// TwinCAT 3 PLC project PDxxPLC
// Title: PDxx
// Company: iMusic AS
// Author: Jakob Bak
// ProjectVersion: 0.4.0.3
// Description: Library for using the Nanotec PDxx series Stepper Motor with Controller
// ProgramVersion: 3.1.4024.0
// libraries:
//   Tc2_Standard, * (Beckhoff Automation GmbH)
//   Tc2_System, * (Beckhoff Automation GmbH)
//   Tc3_Module, * (Beckhoff Automation GmbH)
// project tree:
//   DUTs/ E_PDxx_ErrorNumber.TcDUT, E_PDxx_ModesOfOperation.TcDUT, E_PDxx_State.TcDUT, E_PDxx_TransitionCommand.TcDUT, ST_CANopenDevice.TcDUT, ST_PDxx_ControlWord.TcDUT, ST_PDxx_ErrorRegister.TcDUT, ST_PDxx_IO.TcDUT, ST_PDxx_PredefinedErrorField.TcDUT, ST_PDxx_RxTxPDOs.TcDUT, ST_PDxx_SimulationParameters.TcDUT, ST_PDxx_Status.TcDUT, ST_PDxx_StatusWord.TcDUT
//   / PlcTask.TcTTO
//   POUs/ FB_PDxxSimulation.TcPOU, FB_PDxx.TcPOU, FB_SDO.TcPOU, MAIN.TcPOU, FB_PDxxTester.TcPOU
//   Version/ Global_Version.TcGVL
// real-time tasks:
//   TASK PlcTask: cycle T#10ms, priority 20, ADS port 350
// I/O:
//   DEVICE Device 2 (EtherCAT), AmsNetId 10.3.0.21.3.1
//     Term 1 (EK1100) [EK1100 EtherCAT Coupler (2A E-Bus)]
//       Term 2 (EL6751) [EL6751 CANopen Master]
//       Term 3 (EL9011) [EL9011 End Terminal]
//   DEVICE Device 1 (EL6751), AmsNetId 10.3.0.21.2.1
//     Box 1 (PD2-C411L18-E-65-08)
//     Box 2 (PD4-E601L42-E-65-2)
// variable links:
//   PDxxPLC Instance <-> Device 1 (EL6751)/Box 1 (PD2-C411L18-E-65-08)
//     PlcTask Inputs/MAIN.fbPDxxTester.PDxx.stPDOs.TxPDO_1_6041h_StatusWord <-> TxPDO 1/Inputs/Statusword
//     PlcTask Inputs/MAIN.fbPDxxTester.PDxx.stPDOs.TxPDO_1_6061h_ModesOfOperationDisplay <-> TxPDO 1/Inputs/Modes of operation display
//     PlcTask Inputs/MAIN.fbPDxxTester.PDxx.stPDOs.TxPDO_2_6064h_PositionActualValue <-> TxPDO 2/Inputs/Position actual value
//     PlcTask Inputs/MAIN.fbPDxxTester.PDxx.stPDOs.TxPDO_3_6044h_VelocityActualValue <-> TxPDO 3/Inputs/vl velocity actual value
//     PlcTask Inputs/MAIN.fbPDxxTester.PDxx.stPDOs.TxPDO_4_60FDh_DigitalInputs <-> TxPDO 4/Inputs/Digital Inputs
//     PlcTask Outputs/MAIN.fbPDxxTester.PDxx.stPDOs.RxPDO_1_3202h_MotorDriveSubmodeSelect <-> RxPDO 1/Outputs/Motor drive submode select
//     PlcTask Outputs/MAIN.fbPDxxTester.PDxx.stPDOs.RxPDO_1_6040h_ControlWord <-> RxPDO 1/Outputs/Controlword
//     PlcTask Outputs/MAIN.fbPDxxTester.PDxx.stPDOs.RxPDO_1_6060h_ModesOfOperation <-> RxPDO 1/Outputs/Modes of operation
//     PlcTask Outputs/MAIN.fbPDxxTester.PDxx.stPDOs.RxPDO_2_607Ah_TargetPosition <-> RxPDO 2/Outputs/Target Position
//     PlcTask Outputs/MAIN.fbPDxxTester.PDxx.stPDOs.RxPDO_2_6081h_ProfileVelocity <-> RxPDO 2/Outputs/Profile velocity
//     PlcTask Outputs/MAIN.fbPDxxTester.PDxx.stPDOs.RxPDO_3_6042h_TargetVelocity <-> RxPDO 3/Outputs/vl target velocity
//     PlcTask Outputs/MAIN.fbPDxxTester.PDxx.stPDOs.RxPDO_4_60FEh_DigitalOutputs <-> RxPDO 4/Outputs/Digital Outputs #1

CONFIGURATION PDxxPLC
    RESOURCE PLC ON TwinCAT3
        TASK PlcTask(INTERVAL := T#10ms, PRIORITY := 20);
        PROGRAM MAIN WITH PlcTask : MAIN;
    END_RESOURCE
END_CONFIGURATION

// ---- DUTs/E_PDxx_ErrorNumber.TcDUT
{attribute 'qualified_only'}
{attribute 'strict'}
TYPE E_PDxx_ErrorNumber :
(
	// The following is taken from the manual for the PD4-E(CANopen) section 1003h.
	// It pertains to the firmware version v1748, so other firmware versions and other types of motors may have different error number 
	WATCHDOG_RESET 						:= 0, // Watchdog-Reset
	INPUT_VOLTAGE_TOO_HIGH				:= 1, // Input voltage too high
	OUTPUT_CURRENT_TOO_HIGH 			:= 2, // Output current too high
	INPUT_VOLTAGE_TOO_LOW 				:= 3, // Input voltage too low
	ERROR_AT_FIELDBUS 					:= 4, // Error at fieldbus
	MOTOR_TURNS_WRONG_DIRECTION			:= 5, // Motor turns – in spite of active block – in the wrong direction
	NMT_MASTER_TAKES_TOO_LONG_TO_SEND	:= 6, // CANopen only: NMT master takes too long to send nodeguarding request
	ENCODER_ERROR_ELECTRICAL_FAULT		:= 7, // Encoder error due to electrical fault or defective hardware
	ENCODER_ERROR_INDEX_NOT_FOUND		:= 8, // Encoder error; index not found during the auto setup
	ERROR_IN_AB_TRACK					:= 9, // Error in the AB track
	POSITIVE_LIMIT_SWITCH_ZONE_EXCEEDED := 10, //  Positive limit switch and tolerance zone exceeded
	NEGATIVE_LIMIT_SWITCH_ZONE_EXCEEDED := 11, // Negative limit switch and tolerance zone exceeded
	DEVICE_TEMPERATURE_ERROR			:= 12, // Device temperature above 80°C
	FOLLOWING_ERROR_WINDOW_AND_TIMEOUT	:= 13, // The values of object 6065h (Following Error Window) and object 6066h (Following Error Time Out) were exceeded; a fault was triggered.
	NONVOLATIVE_MEMORY_FULL_FOURTEEN	:= 14, // Warning: Nonvolatile memory full; controller must be restarted for cleanup work.
	MOTOR_BLOCKED						:= 15, // Motor blocked
	NONVOLATIVE_MEMORY_DAMAGED			:= 16, // Warning: Nonvolatile memory damaged; controller must be restarted for cleanup work.
	SLAVE_TOOK_TOO_LONG_TO_SEND_PDO		:= 17, // CANopen only: Slave took too long TO send PDO messages.
	HALL_SENSOR_FAULTY					:= 18, // Hall sensor faulty
	PDO_NOT_PROCESSED_DUE_LENGTH_ERROR	:= 19, // CANopen only: PDO not processed due to a length error
	PDO_LENGTH_EXCEEDED					:= 20, // CANopen only: PDO length exceeded
	NONVOLATIVE_MEMORY_FULL_TWENTY_ONE	:= 21, // Warning: Nonvolatile memory full; controller must be restarted for cleanup work.
	RATED_CURRENT_MUST_BE_SET			:= 22, // Rated current must be set (203Bh:01h)
	ENCODER_RESOLUTION_SET_INCORRECTLY	:= 23, // Encoder resolution, number of pole pairs and some other values are incorrect.
	MOTOR_CURRENT_TOO_HIGH_ADJUST_PI	:= 24, // Motor current is too high, adjust the PI parameters.
	INTERNAL_SOFTWARE_ERROR				:= 25, // Internal software error, generic
	CURRENT_TOO_HIGH_AT_DIGITAL_OUTPUT	:= 26, // Current too high at digital output
	UNEXPECTED_SYNC_LENGTH				:= 27, // CANopen only: Unexpected sync length
	OP_SWITCH_WITHOUT_STOPPING_MOTOR	:= 28, // EtherCAT only: The motor was stopped because EtherCAT switched state from OP to either SafeOP or PreOP without first stopping the motor.
	SLIPPAGE_ERROR_TOO_LARGE			:= 30 // Error in speed monitoring: slippage error too large
);
END_TYPE

// ---- DUTs/E_PDxx_ModesOfOperation.TcDUT
{attribute 'qualified_only'}
{attribute 'strict'}
TYPE E_PDxx_ModesOfOperation :
(
	AUTO_SETUP := -2,
	CLOCK_DIRECTION_MODE,
	NO_MODE_CHANGE_OR_NO_MODE_ASSIGNED,
	PROFILE_POSITION_MODE,
	VELOCITY_MODE,
	PROFILE_VELOCITY_MODE,
	PROFILE_TORQUE_MODE,
	RESERVED,
	HOMING_MODE,
	INTERPOLATED_POSITION_MODE,
	CYCLIC_SYNCHRONOUS_POSITION_MODE,
	CYCLIC_SYNCHRONOUS_VELOCITY_MODE,
	CYCLIC_SYNCHRONOUS_TORQUE_MODE
);
END_TYPE

// ---- DUTs/E_PDxx_State.TcDUT
{attribute 'qualified_only'}
{attribute 'strict'}
TYPE E_PDxx_State :
(
	UNKNOWN_STATE, 
	NOT_READY_TO_SWITCH_ON, 
	SWITCH_ON_DISABLED, 
	READY_TO_SWITCH_ON, 
	SWITCHED_ON, 
	OPERATION_ENABLED, 
	QUICK_STOP_ACTIVE, 
	FAULT_REACTION_ACTIVE, 
	FAULT
);
END_TYPE

// ---- DUTs/E_PDxx_TransitionCommand.TcDUT
{attribute 'qualified_only'}
{attribute 'strict'}
TYPE E_PDxx_TransitionCommand :
(
	SHUTDOWN := 0,
	SWITCH_ON,
	DISABLE_VOLTAGE,
	QUICK_STOP,
	ENABLE_OPERATION,
	FAULT_RESET
);
END_TYPE

// ---- DUTs/ST_CANopenDevice.TcDUT
TYPE ST_CANopenDevice :
STRUCT
    AmsNetId	: STRING(23); (* The AMSNetID addresses the EL6751. Can be empty if only one local single channel card is present*)
    PortNr		: WORD;       (* This Port No. addresses the CANopen Node (see System Manager) *)
END_STRUCT
END_TYPE

// ---- DUTs/ST_PDxx_ControlWord.TcDUT
TYPE ST_PDxx_ControlWord :
STRUCT
	SwitchedOn_bit_0			: BOOL; // Value = "1": Switches to the "Switched on" state
	EnableVoltage_bit_1			: BOOL; // Value = "1": Switches to the "Enable voltage" state
	QuickStop_bit_2				: BOOL; // Value = "0": Switches to the "Quick stop" state
	EnableOperation_bit_3		: BOOL; // Value = "1": Switches to the "Enable operation" state
	OperationModeSpecific_bit_4	: BOOL; // Meaning is dependent on the selected operating mode
	OperationModeSpecific_bit_5	: BOOL; // Meaning is dependent on the selected operating mode
	OperationModeSpecific_bit_6	: BOOL; // Meaning is dependent on the selected operating mode
	FaultReset_bit_7			: BOOL; // Resets an error (if possible)
	Halt_bit_8					: BOOL; // Value = "1": Triggers a halt; valid in the following modes: Profile Position, Velocity, Profile Velocity, Profile Torque, Interpolated Position Mode
	OperationModeSpecific_bit_9	: BOOL; // not described in the manual...
	
	eState : E_PDxx_State;
END_STRUCT
END_TYPE

// ---- DUTs/ST_PDxx_ErrorRegister.TcDUT

TYPE ST_PDxx_ErrorRegister :
STRUCT
	// Taken from manual section "1001h Error Register"
	GEN : BIT; // bit 0 - General error
	CUR : BIT; // bit 1 - Current
	VOL : BIT; // bit 2 - Voltage
	TEMP: BIT; // bit 3 - Temperature
	COM : BIT; // bit 4 - Communication
	PROF: BIT; // bit 5 - Relates TO the device profile
	RES : BIT; // bit 6 - Reserved, always "0"
	MAN : BIT; // bit 7 - Manufacturer-specific: The motor turns in the wrong direction.
END_STRUCT
END_TYPE

// ---- DUTs/ST_PDxx_IO.TcDUT
TYPE ST_PDxx_IO :
STRUCT
(* These values can be read with PDO on 60FDh *)
	InputNegativeLimitSwitch		: BOOL;
	InputPositiveLimitSwitch		: BOOL;
	InputHomeSwitch					: BOOL;
	Input1		: BOOL;
	Input2		: BOOL;
	Input3		: BOOL;
	Input4		: BOOL;
	Input5		: BOOL;
	Input6		: BOOL;
	Input7		: BOOL;
	Input8		: BOOL;

(* The below values has to be read/set with SDO 3240h *)	
	InputNegativeLimitSwitchEnabled	: BOOL;
	InputPositiveLimitSwitchEnabled	: BOOL;
	InputHomeSwitchEnabled			: BOOL;
	Input1_Inverted	: BOOL;
	Input2_Inverted	: BOOL;
	Input3_Inverted	: BOOL;
	Input4_Inverted	: BOOL;
	Input5_Inverted	: BOOL;
	Input6_Inverted	: BOOL;
	Input7_Inverted	: BOOL;
	Input8_Inverted	: BOOL;
	Input1_24V		: BOOL;
	Input2_24V		: BOOL;
	Input3_24V		: BOOL;
	Input4_24V		: BOOL;
	Input5_24V		: BOOL;
	Input6_24V		: BOOL;
	Input7_24V		: BOOL;
	Input8_24V		: BOOL;

//	OutputBrake	: BOOL;
//	Output1		: BOOL;
//	Output2		: BOOL;
//	Output3		: BOOL;
//	Output4		: BOOL;
END_STRUCT
END_TYPE

// ---- DUTs/ST_PDxx_PredefinedErrorField.TcDUT

TYPE ST_PDxx_PredefinedErrorField :
STRUCT
	nErrorNumber	: USINT;
	stErrorClass	: ST_PDxx_ErrorRegister;
	nErrorCode		: UINT;
END_STRUCT
END_TYPE

// ---- DUTs/ST_PDxx_RxTxPDOs.TcDUT
TYPE ST_PDxx_RxTxPDOs :
STRUCT
	TxPDO_1_6041h_StatusWord					: UINT;
	TxPDO_1_6061h_ModesOfOperationDisplay		: SINT;
	TxPDO_2_6064h_PositionActualValue			: DINT;
	TxPDO_3_6044h_VelocityActualValue			: INT;
	TxPDO_4_60FDh_DigitalInputs					: UDINT;
	
	RxPDO_1_6040h_ControlWord					: UINT;
	RxPDO_1_6060h_ModesOfOperation				: SINT;
	RxPDO_1_3202h_MotorDriveSubmodeSelect		: UDINT;
	RxPDO_2_607Ah_TargetPosition				: DINT;
	RxPDO_2_6081h_ProfileVelocity				: UDINT;
	RxPDO_3_6042h_TargetVelocity				: INT;
	RxPDO_4_60FEh_DigitalOutputs				: UDINT;
END_STRUCT
END_TYPE

// ---- DUTs/ST_PDxx_SimulationParameters.TcDUT
TYPE ST_PDxx_SimulationParameters :
STRUCT
	bActivateSimulation		: BOOL := FALSE;
	nPositionMin			: LREAL := 0; // mm
	nPositionMax			: LREAL := 1000; // mm
	nSecondsPerSimStep 		: LREAL := 0.010; // seconds
	nMMPerSecondPerVelUnit	: LREAL := 0.1667; // mm/s, for example rpm at 10mm per revolution, is 10 mm per minute, and hence this value 10 / 60 = 0.16667.
	
	bObjectInserted			: BOOL;
	nObjectThickness		: LREAL := 0.0; // mm
END_STRUCT
END_TYPE

// ---- DUTs/ST_PDxx_Status.TcDUT
TYPE ST_PDxx_Status :
STRUCT
	bZeroInitialised 			: BOOL := FALSE;
	bReversePolarity			: BOOL;
	nHomePosition				: DINT;
	nCurrentPosition			: DINT;
	nCurrentVelocity			: INT;
	nTargetPosition				: DINT;
	nMinActualPosition			: DINT;
	nMaxActualPosition			: DINT;
	bHasError					: BOOL;
	stErrorRegister				: ST_PDxx_ErrorRegister;
	nNumErrors					: USINT;
	ErrorField					: ARRAY [1..8] OF ST_PDxx_PredefinedErrorField;
END_STRUCT
END_TYPE

// ---- DUTs/ST_PDxx_StatusWord.TcDUT
TYPE ST_PDxx_StatusWord :
STRUCT
	ReadyToSwitchOn		: BOOL; // Value = "1": Controller is in the "Ready to Switch On" state (dependent on other bits, see following bit mask)
	SwitchedOn 			: BOOL; // Value = "1": Controller is in the "Switched On" state (dependent on other bits, see following bit mask)
	OperationEnabled	: BOOL; // Value = "1": Controller is in the "Operation Enabled" state (dependent on other bits, see following bit mask)
	Fault				: BOOL; // Error occurred
	VoltageEnabled		: BOOL; // Voltage applied
	QuickStop			: BOOL; // Value = "0": Controller is in the "Quick Stop" state (dependent on other bits, see following bit mask)
	SwitchOnDisabled	: BOOL;	// Value = "1": Controller is in the "Switched On Disabled" state (dependent on other bits, see following bit mask)
	Warning				: BOOL;	// Value = "1": Warning
	Synchronization		: BOOL;	// Value = "1": Controller is in sync with the fieldbus; value = "0": Controller is not in sync with the fieldbus
	Remote				: BOOL;	// Remote (value of the bit is always "1")
	TargetReached		: BOOL; // Target reached
	InternalLimitReached: BOOL;	// Limit exceeded
	OperationModeSpecific_bit12: BOOL; // Meaning is dependent on the selected operating mode
	OperationModeSpecific_bit13: BOOL; // Meaning is dependent on the selected operating mode
	ClosedLoopAvailable	: BOOL; // Value = "1": Auto setup was successful and encoder index seen: closed loop mode possible
END_STRUCT
END_TYPE

// ---- Version/Global_Version.TcGVL
{attribute 'TcGenerated'}
{attribute 'no-analysis'}
{attribute 'linkalways'}
// This function has been automatically generated from the project information.
VAR_GLOBAL CONSTANT
	{attribute 'const_non_replaced'}
	stLibVersion_PDxx : ST_LibVersion := (iMajor := 0, iMinor := 4, iBuild := 0, iRevision := 3, nFlags := 1, sVersion := '0.4.0.3');
END_VAR

// ---- POUs/MAIN.TcPOU

PROGRAM MAIN
VAR
	fbPDxxTester : FB_PDxxTester;
	stCANopenDevice : ST_CANopenDevice := (AmsNetId:='10.3.0.21.2.1', PortNr := 16#1001);
END_VAR


fbPDxxTester(stCANopenDevice := stCANopenDevice);

END_PROGRAM

// ---- POUs/FB_PDxxTester.TcPOU

FUNCTION_BLOCK FB_PDxxTester
VAR_INPUT

	stCANopenDevice 	: ST_CANopenDevice;
//	SimParameters		: ST_PDxx_SimulationParameters;
//	bStandAloneTesting 	: BOOL 		:= FALSE;

	nTargetVelocity		: INT := 100;			// what unit ?
	nTargetPosition		: DINT := 0;		// what unit ?
	nTargetCurrent		: UDINT := 1000;	// mA ?
//	bExecuteMove		: BOOL  := FALSE;
	
	nFeedRate			: UDINT := 44533;
	nFeedRateDivisor	: UDINT	:= 2000;
	nZeroingMaxCurrent	: UDINT := 1000;
	bReversePolarity	: BOOL := FALSE;
	
	eMode : (NO_CHANGE := 0, RESET, HOME, POSITION, VELOCITY);
END_VAR

VAR_OUTPUT
//	bTargetPositionReceived: BOOL;
	eState				: E_PDxx_State;
	eModesOfOperation	: E_PDxx_ModesOfOperation;
	
	Status 				: ST_PDxx_Status;
	StateEntryTime		: TIME;
	bStateComplete		: BOOL;
END_VAR

VAR
	PDxx : FB_PDxx;
//	trExecute : R_TRIG;
	eLastMode 			: INT;
END_VAR


ExecuteState();

PDxx(
	stCANopenDevice := stCANopenDevice,
//	SimParameters := SimParameters,
//	bStandAloneTesting := bStandAloneTesting,
//	bStandAloneTestSendTarget := bExecuteMove,
//	bStandAloneTestSendTargetSuccess => bTargetPositionReceived,
	Status => Status
);

eState := PDxx.eState;
eModesOfOperation := PDxx.eModesOfOperation;


METHOD PRIVATE ExecuteState

IF eMode <> NO_CHANGE THEN
	IF eMode <> eLastMode THEN
		eLastMode := eMode;
		StateEntryTime := TIME();
		bStateComplete := FALSE;
	END_IF
	
//	trExecute(CLK := bExecuteMove);	
	
	CASE eMode OF

		RESET:
			M_Resetting();

		HOME:
			PDxx.ProbeActualPositionLimits(nTargetVelocity);

		POSITION:
//			IF trExecute.Q = TRUE THEN
				PDxx.GoToTargetPosition(nPosition := nTargetPosition, nVelocity := nTargetVelocity, nMaxCurrent := nTargetCurrent);		
//			END_IF

		VELOCITY:
//			IF trExecute.Q = TRUE THEN
				PDxx.GoToTargetVelocity(nVelocity := nTargetVelocity, nMaxCurrent := nTargetCurrent);		
//			END_IF		

	END_CASE
	
	IF bStateComplete THEN
		eMode := NO_CHANGE;
	END_IF

END_IF
END_METHOD


METHOD PRIVATE M_Resetting : BOOL
VAR
	bFeedRateSetpointReached 	: BOOL := FALSE;
	bMaxCurrentSetpointReached 	: BOOL := FALSE;
	bPolaritySetpointReached	: BOOL := FALSE;
END_VAR

IF PDxx.SetFeedRate(nFeedRate := nFeedRate, nDivisor := nFeedRateDivisor) THEN
	bFeedRateSetpointReached := TRUE;
END_IF

IF PDxx.fbSdoMaxCurrentValue = nZeroingMaxCurrent THEN
	bMaxCurrentSetpointReached := TRUE;
ELSE
	PDxx.SetMaxCurrent(nZeroingMaxCurrent);
END_IF

IF 	PDxx.IsPolarityReversed() = bReversePolarity THEN
	bPolaritySetpointReached := TRUE;
ELSE
	bPolaritySetpointReached := PDxx.SetReversePolarity(bReversePolarity);
END_IF

(* COMPLETE STATE *)
IF 	bFeedRateSetpointReached AND
	bMaxCurrentSetpointReached AND
	bPolaritySetpointReached THEN 
	IF PDxx.SwitchOnPowerToMotor() THEN
		bStateComplete := TRUE;
	END_IF
ELSE
	PDxx.SwitchOffPowerToMotor();
END_IF
END_METHOD

END_FUNCTION_BLOCK

// ---- POUs/FB_PDxx.TcPOU
FUNCTION_BLOCK FB_PDxx

VAR_INPUT
	SimParameters		: ST_PDxx_SimulationParameters;

	eState				: E_PDxx_State;
	eModesOfOperation	: E_PDxx_ModesOfOperation;

	bStandAloneTesting 				: BOOL 		:= FALSE;
	eStandAloneTestState			: E_PDxx_State;
	eStandAloneTestModesOfOperation	: E_PDxx_ModesOfOperation;
	bStandAloneTestSendTarget		: BOOL 		:= 0;
	
	stCANopenDevice : ST_CANopenDevice;

	fbSdoErrorRegister				: FB_SDO	:= (CO_Index:=16#1001, CO_SubIndex:=16#0, DataLength:=1, 	CO_Name:='Error Register', 			stCANopenDevice:=stCANopenDevice);
	fbSdoErrorRegisterValue 		: USINT;

	fbSdoNumberOfErrors				: FB_SDO	:= (CO_Index:=16#1003, CO_SubIndex:=16#0, DataLength:=1, 	CO_Name:='Number Of Errors', 		stCANopenDevice:=stCANopenDevice);
	fbSdoNumberOfErrorsValue 		: USINT;

	fbSdoErrorField_1				: FB_SDO	:= (CO_Index:=16#1003, CO_SubIndex:=16#1, DataLength:=4, 	CO_Name:='Standard Error Field 1', 	stCANopenDevice:=stCANopenDevice);
	fbSdoErrorField_2				: FB_SDO	:= (CO_Index:=16#1003, CO_SubIndex:=16#2, DataLength:=4, 	CO_Name:='Standard Error Field 2', 	stCANopenDevice:=stCANopenDevice);
	fbSdoErrorField_3				: FB_SDO	:= (CO_Index:=16#1003, CO_SubIndex:=16#3, DataLength:=4, 	CO_Name:='Standard Error Field 3', 	stCANopenDevice:=stCANopenDevice);
	fbSdoErrorField_4				: FB_SDO	:= (CO_Index:=16#1003, CO_SubIndex:=16#4, DataLength:=4, 	CO_Name:='Standard Error Field 4', 	stCANopenDevice:=stCANopenDevice);
	fbSdoErrorField_5				: FB_SDO	:= (CO_Index:=16#1003, CO_SubIndex:=16#5, DataLength:=4, 	CO_Name:='Standard Error Field 5', 	stCANopenDevice:=stCANopenDevice);
	fbSdoErrorField_6				: FB_SDO	:= (CO_Index:=16#1003, CO_SubIndex:=16#6, DataLength:=4, 	CO_Name:='Standard Error Field 6', 	stCANopenDevice:=stCANopenDevice);
	fbSdoErrorField_7				: FB_SDO	:= (CO_Index:=16#1003, CO_SubIndex:=16#7, DataLength:=4, 	CO_Name:='Standard Error Field 7', 	stCANopenDevice:=stCANopenDevice);
	fbSdoErrorField_8				: FB_SDO	:= (CO_Index:=16#1003, CO_SubIndex:=16#8, DataLength:=4, 	CO_Name:='Standard Error Field 8', 	stCANopenDevice:=stCANopenDevice);
	fbSdoErrorFieldValue			: ARRAY [1..8] OF UDINT;

	fbSdoMaxCurrent					: FB_SDO	:= (CO_Index:=16#2031, CO_SubIndex:=16#0, DataLength:=4, 	CO_Name:='Maximum Current', 		stCANopenDevice:=stCANopenDevice);
	fbSdoMaxCurrentValue 			: UDINT;

//	fbSdoPolarity					: FB_SDO	:= (CO_Index:=16#607E, CO_SubIndex:=16#0, DataLength:=1, 	CO_Name:='Polarity', 				stCANopenDevice:=fbEL6751);
//	fbSdoPolarityValue				: USINT;

	fbSdoSpecialFunctionEnable		: FB_SDO	:= (CO_Index:=16#3040, CO_SubIndex:=16#1, DataLength:=4, 	CO_Name:='Special Function Enable',	stCANopenDevice:=stCANopenDevice);
	fbSdoSpecialFunctionEnableValue	: UDINT;

	fbSdoFunctionInverted			: FB_SDO	:= (CO_Index:=16#3040, CO_SubIndex:=16#2, DataLength:=4, 	CO_Name:='Function Inverted',		stCANopenDevice:=stCANopenDevice);
	fbSdoFunctionInvertedValue		: UDINT;
	
	fbSdoInputRangeSelect			: FB_SDO	:= (CO_Index:=16#3040, CO_SubIndex:=16#6, DataLength:=4, 	CO_Name:='Input Range Select',		stCANopenDevice:=stCANopenDevice);
	fbSdoInputRangeSelectValue		: UDINT;
	
	fbSdoFeed						: FB_SDO	:= (CO_Index:=16#6092, CO_SubIndex:=16#1, DataLength:=4, 	CO_Name:='Feed', 					stCANopenDevice:=stCANopenDevice);
	fbSdoFeedValue					: UDINT;

	fbSdoShaftRevolutions			: FB_SDO	:= (CO_Index:=16#6092, CO_SubIndex:=16#2, DataLength:=4, 	CO_Name:='Shaft Revolutions', 		stCANopenDevice:=stCANopenDevice);
	fbSdoShaftRevolutionsValue		: UDINT;
	
	fbSdoEncoderIncrements			: FB_SDO	:= (CO_Index:=16#608F, CO_SubIndex:=16#1, DataLength:=4, 	CO_Name:='Encoder Increments', 		stCANopenDevice:=stCANopenDevice);
	fbSdoEncoderIncrementsValue		: UDINT;

	fbSdoMotorRevolutions			: FB_SDO	:= (CO_Index:=16#608F, CO_SubIndex:=16#2, DataLength:=4, 	CO_Name:='Motor Revolutions', 		stCANopenDevice:=stCANopenDevice);
	fbSdoMotorRevolutionsValue		: UDINT;
	
	fbSdoSIUnitPosition				: FB_SDO	:= (CO_Index:=16#60A8, CO_SubIndex:=16#0, DataLength:=4, 	CO_Name:='SI Unit Position', 		stCANopenDevice:=stCANopenDevice);
	fbSdoSIUnitPositionValue		: UDINT;
	
	fbSdoProfileAcceleration		: FB_SDO	:= (CO_Index:=16#6083, CO_SubIndex:=16#0, DataLength:=4, 	CO_Name:='Profile Acceleration', 	stCANopenDevice:=stCANopenDevice);
	fbSdoProfileAccelerationValue	: UDINT;

	fbSdoProfileDeceleration		: FB_SDO	:= (CO_Index:=16#6084, CO_SubIndex:=16#0, DataLength:=4, 	CO_Name:='Profile Deceleration', 	stCANopenDevice:=stCANopenDevice);
	fbSdoProfileDecelerationValue	: UDINT;

END_VAR

VAR_OUTPUT
	Status						: ST_PDxx_Status;
	bStandAloneTestSendTargetSuccess: BOOL;
END_VAR

VAR
	stPDOs : ST_PDxx_RxTxPDOs := (
		RxPDO_1_3202h_MotorDriveSubmodeSelect 	:= 16#00000001, // default to closed loop
		RxPDO_2_6081h_ProfileVelocity 			:= 16#000001F4 // default to 500 RPM
	);
	
	stIO : ST_PDxx_IO;
	
	stStatusWord : ST_PDxx_StatusWord;
	stControlWord : ST_PDxx_ControlWord;

	Simulate			: FB_PDxxSimulation;
	
END_VAR


CheckForErrors();
CheckState();
CheckModesOfOperation();
CheckDigitalInputs();
ResetControlWordBit4();

IF SimParameters.bActivateSimulation = TRUE THEN
	Simulate(
		Parameters								:= SimParameters,
		RxPDO_1_6040h_ControlWord  				:= stPDOs.RxPDO_1_6040h_ControlWord,
		RxPDO_1_6060h_ModesOfOperation  		:= stPDOs.RxPDO_1_6060h_ModesOfOperation,
		RxPDO_1_3202h_MotorDriveSubmodeSelect  	:= stPDOs.RxPDO_1_3202h_MotorDriveSubmodeSelect,
		RxPDO_2_607Ah_TargetPosition  			:= stPDOs.RxPDO_2_607Ah_TargetPosition,
		RxPDO_2_6081h_ProfileVelocity			:= stPDOs.RxPDO_2_6081h_ProfileVelocity,
		RxPDO_3_6042h_TargetVelocity			:= stPDOs.RxPDO_3_6042h_TargetVelocity,
		RxPDO_4_60FEh_DigitalOutputs			:= stPDOs.RxPDO_4_60FEh_DigitalOutputs);
		
	stPDOs.TxPDO_1_6041h_StatusWord 				:= Simulate.TxPDO_1_6041h_StatusWord;
	stPDOs.TxPDO_1_6061h_ModesOfOperationDisplay	:= Simulate.TxPDO_1_6061h_ModesOfOperationDisplay;
	stPDOs.TxPDO_2_6064h_PositionActualValue		:= Simulate.TxPDO_2_6064h_PositionActualValue;
	stPDOs.TxPDO_3_6044h_VelocityActualValue		:= Simulate.TxPDO_3_6044h_VelocityActualValue;
	stPDOs.TxPDO_4_60FDh_DigitalInputs				:= Simulate.TxPDO_4_60FDh_DigitalInputs;
END_IF

IF bStandAloneTesting = TRUE THEN
	IF eModesOfOperation <> eStandAloneTestModesOfOperation THEN
		ChangeModesOfOperation(eModesOfOperation := eStandAloneTestModesOfOperation);
	END_IF
	
	IF eState <> eStandAloneTestState THEN
		ChangeState(eRequestedState := eStandAloneTestState);
	END_IF
	
	IF bStandAloneTestSendTarget THEN
		bStandAloneTestSendTargetSuccess := StartMoveToTargetPosition();
		bStandAloneTestSendTarget := FALSE;
	END_IF	
END_IF

ACTION Abort:

IF SwitchOffPowerToMotor() = TRUE THEN
	ResetStatusAndSDOs();
END_IF
END_ACTION

METHOD ChangeModesOfOperation : BOOL
VAR_INPUT
	eModesOfOperation : E_PDxx_ModesOfOperation;
END_VAR
VAR
	ModesOfOperation : SINT;
END_VAR
CASE eModesOfOperation OF
	
	E_PDxx_ModesOfOperation.AUTO_SETUP:
		ModesOfOperation := -2;
	E_PDxx_ModesOfOperation.CLOCK_DIRECTION_MODE:
		ModesOfOperation := -1;
	E_PDxx_ModesOfOperation.NO_MODE_CHANGE_OR_NO_MODE_ASSIGNED:
		ModesOfOperation := 0;
	E_PDxx_ModesOfOperation.PROFILE_POSITION_MODE:
		ModesOfOperation := 1;
	E_PDxx_ModesOfOperation.VELOCITY_MODE:
		ModesOfOperation := 2;
	E_PDxx_ModesOfOperation.PROFILE_VELOCITY_MODE:
		ModesOfOperation := 3;
	E_PDxx_ModesOfOperation.PROFILE_TORQUE_MODE:
		ModesOfOperation := 4;
	E_PDxx_ModesOfOperation.RESERVED:
		ModesOfOperation := 5;
	E_PDxx_ModesOfOperation.HOMING_MODE:
		ModesOfOperation := 6;
	E_PDxx_ModesOfOperation.INTERPOLATED_POSITION_MODE:
		ModesOfOperation := 7;
	E_PDxx_ModesOfOperation.CYCLIC_SYNCHRONOUS_POSITION_MODE:
		ModesOfOperation := 8;
	E_PDxx_ModesOfOperation.CYCLIC_SYNCHRONOUS_VELOCITY_MODE:
		ModesOfOperation := 9;
	E_PDxx_ModesOfOperation.CYCLIC_SYNCHRONOUS_TORQUE_MODE:	
		ModesOfOperation := 10;
ELSE
	ChangeModesOfOperation := FALSE;
	RETURN;

END_CASE

stPDOs.RxPDO_1_6060h_ModesOfOperation := ModesOfOperation;
ChangeModesOfOperation := TRUE;
END_METHOD

METHOD ChangeState : BOOL
VAR_INPUT
	eRequestedState : E_PDxx_State; 
END_VAR
VAR
	ControlWord : UINT;
END_VAR
VAR_INST
	bLastFaultResetBitState : BOOL;
END_VAR

ControlWord := 0;

IF eState = E_PDxx_State.FAULT THEN
	IF Status.bHasError = FALSE THEN
		bLastFaultResetBitState := bLastFaultResetBitState XOR 1; 
		stControlWord.FaultReset_bit_7	:= bLastFaultResetBitState;	// "Fault reset" transition 13 on rising edge
	ELSE
		stControlWord.FaultReset_bit_7 := FALSE;	// "Fault reset" transition 13 on rising edge		
	END_IF
	ControlWord.7 := stControlWord.FaultReset_bit_7;
	stPDOs.RxPDO_1_6040h_ControlWord := ControlWord;
	RETURN;
END_IF

(* All of the below cases are taken from the transistion diagram on p. 34 in the manual *)

CASE eRequestedState OF

	// E_PD2C_State.NOT_READY_TO_SWITCH_ON:
		// Can not be triggered from software

	E_PDxx_State.SWITCH_ON_DISABLED: 			// "Disable Voltage" transitions 6, 7, 9, 12 
		stControlWord.EnableVoltage_bit_1	:= FALSE;
		stControlWord.FaultReset_bit_7		:= FALSE;
		
	E_PDxx_State.READY_TO_SWITCH_ON: 			// "Shutdown" transitions 1, 5, 8 
		stControlWord.SwitchedOn_bit_0		:= FALSE;
		stControlWord.EnableVoltage_bit_1	:= TRUE;
		stControlWord.QuickStop_bit_2		:= TRUE; // Quick stop is Active Low
		stControlWord.FaultReset_bit_7		:= FALSE;

	E_PDxx_State.SWITCHED_ON:					// "Switch On" and "Diable operation" transitions 2, 4 
		stControlWord.SwitchedOn_bit_0		:= TRUE;
		stControlWord.EnableVoltage_bit_1	:= TRUE;
		stControlWord.QuickStop_bit_2		:= TRUE; // Quick stop is Active Low
		stControlWord.EnableOperation_bit_3	:= FALSE;
		stControlWord.FaultReset_bit_7		:= FALSE;

	E_PDxx_State.OPERATION_ENABLED: 				// "Enable operation" transition 3
		stControlWord.SwitchedOn_bit_0		:= TRUE;
		stControlWord.EnableVoltage_bit_1	:= TRUE;
		stControlWord.QuickStop_bit_2		:= TRUE; // Quick stop is Active Low
		stControlWord.EnableOperation_bit_3	:= TRUE;
		stControlWord.FaultReset_bit_7		:= FALSE;

	E_PDxx_State.QUICK_STOP_ACTIVE: 				// "Quick stop" transition 10 
		stControlWord.EnableVoltage_bit_1	:= TRUE;
		stControlWord.QuickStop_bit_2		:= FALSE; // Quick stop is Active Low
		stControlWord.FaultReset_bit_7		:= FALSE;

	// E_PD2C_State.FAULT_REACTION_ACTIVE:
		// Can not be triggered by software
	// E_PD2C_State.FAULT:
		// Can not be triggered by software

END_CASE

stControlWord.eState						:= eRequestedState;

ControlWord.0 := stControlWord.SwitchedOn_bit_0;
ControlWord.1 := stControlWord.EnableVoltage_bit_1;
ControlWord.2 := stControlWord.QuickStop_bit_2;
ControlWord.3 := stControlWord.EnableOperation_bit_3;
ControlWord.4 := stControlWord.OperationModeSpecific_bit_4;
ControlWord.5 := stControlWord.OperationModeSpecific_bit_5;
ControlWord.6 := stControlWord.OperationModeSpecific_bit_6;
ControlWord.7 := stControlWord.FaultReset_bit_7;
ControlWord.8 := stControlWord.Halt_bit_8;
ControlWord.9 := stControlWord.OperationModeSpecific_bit_9;

stPDOs.RxPDO_1_6040h_ControlWord := ControlWord;
END_METHOD

METHOD PUBLIC CheckDigitalInputs
VAR
	i : UINT;
END_VAR
stIO.InputNegativeLimitSwitch	:= stPDOs.TxPDO_4_60FDh_DigitalInputs.1;
stIO.InputPositiveLimitSwitch	:= stPDOs.TxPDO_4_60FDh_DigitalInputs.2;
stIO.InputHomeSwitch			:= stPDOs.TxPDO_4_60FDh_DigitalInputs.3;
stIO.Input1 := stPDOs.TxPDO_4_60FDh_DigitalInputs.16;
stIO.Input2 := stPDOs.TxPDO_4_60FDh_DigitalInputs.17;
stIO.Input3 := stPDOs.TxPDO_4_60FDh_DigitalInputs.18;
stIO.Input4 := stPDOs.TxPDO_4_60FDh_DigitalInputs.19;
stIO.Input5 := stPDOs.TxPDO_4_60FDh_DigitalInputs.20;
stIO.Input6 := stPDOs.TxPDO_4_60FDh_DigitalInputs.21;
stIO.Input7 := stPDOs.TxPDO_4_60FDh_DigitalInputs.22;
stIO.Input8 := stPDOs.TxPDO_4_60FDh_DigitalInputs.23;
END_METHOD

ACTION CheckForErrors:

fbSdoErrorRegister(bStartReading := TRUE);
IF fbSdoErrorRegister.ReadDataAvailable THEN
	fbSdoErrorRegisterValue := fbSdoErrorRegister.GetReadDataAsUSINT();
	Status.bHasError := fbSdoErrorRegisterValue <> 0;
	Status.stErrorRegister := ParseErrorRegister(fbSdoErrorRegisterValue);
END_IF

fbSdoNumberOfErrors(bStartReading := TRUE);
IF fbSdoNumberOfErrors.ReadDataAvailable THEN
	fbSdoNumberOfErrorsValue := fbSdoNumberOfErrors.GetReadDataAsUSINT();
	Status.nNumErrors := fbSdoNumberOfErrorsValue;
END_IF

// Check for error field 1
IF Status.nNumErrors >= 1 THEN
	fbSdoErrorField_1(bStartReading := TRUE);
	IF fbSdoErrorField_1.ReadDataAvailable THEN
		fbSdoErrorFieldValue[1] := fbSdoErrorField_1.GetReadDataAsUDINT();
		Status.ErrorField[1] := ParseErrorField(fbSdoErrorFieldValue[1]);
	END_IF
ELSE
	fbSdoErrorFieldValue[1] := 0;
	Status.ErrorField[1] := ParseErrorField(fbSdoErrorFieldValue[1]);		
END_IF

// Check for error field 2
IF Status.nNumErrors >= 2 THEN
	fbSdoErrorField_2(bStartReading := TRUE);
	IF fbSdoErrorField_2.ReadDataAvailable THEN
		fbSdoErrorFieldValue[2] := fbSdoErrorField_2.GetReadDataAsUDINT();
		Status.ErrorField[2] := ParseErrorField(fbSdoErrorFieldValue[2]);
	END_IF
ELSE
	fbSdoErrorFieldValue[2] := 0;
	Status.ErrorField[2] := ParseErrorField(fbSdoErrorFieldValue[2]);		
END_IF

// Check for error field 3
IF Status.nNumErrors >= 3 THEN
	fbSdoErrorField_3(bStartReading := TRUE);
	IF fbSdoErrorField_3.ReadDataAvailable THEN
		fbSdoErrorFieldValue[3] := fbSdoErrorField_3.GetReadDataAsUDINT();
		Status.ErrorField[3] := ParseErrorField(fbSdoErrorFieldValue[3]);
	END_IF
ELSE
	fbSdoErrorFieldValue[3] := 0;
	Status.ErrorField[3] := ParseErrorField(fbSdoErrorFieldValue[3]);		
END_IF

// Check for error field 4
IF Status.nNumErrors >= 4 THEN
	fbSdoErrorField_4(bStartReading := TRUE);
	IF fbSdoErrorField_4.ReadDataAvailable THEN
		fbSdoErrorFieldValue[4] := fbSdoErrorField_4.GetReadDataAsUDINT();
		Status.ErrorField[4] := ParseErrorField(fbSdoErrorFieldValue[4]);
	END_IF
ELSE
	fbSdoErrorFieldValue[4] := 0;
	Status.ErrorField[4] := ParseErrorField(fbSdoErrorFieldValue[4]);		
END_IF

// Check for error field 5
IF Status.nNumErrors >= 5 THEN
	fbSdoErrorField_5(bStartReading := TRUE);
	IF fbSdoErrorField_5.ReadDataAvailable THEN
		fbSdoErrorFieldValue[5] := fbSdoErrorField_5.GetReadDataAsUDINT();
		Status.ErrorField[5] := ParseErrorField(fbSdoErrorFieldValue[5]);
	END_IF
ELSE
	fbSdoErrorFieldValue[5] := 0;
	Status.ErrorField[5] := ParseErrorField(fbSdoErrorFieldValue[5]);		
END_IF

// Check for error field 6
IF Status.nNumErrors >= 6 THEN
	fbSdoErrorField_6(bStartReading := TRUE);
	IF fbSdoErrorField_6.ReadDataAvailable THEN
		fbSdoErrorFieldValue[6] := fbSdoErrorField_6.GetReadDataAsUDINT();
		Status.ErrorField[6] := ParseErrorField(fbSdoErrorFieldValue[6]);
	END_IF
ELSE
	fbSdoErrorFieldValue[6] := 0;
	Status.ErrorField[6] := ParseErrorField(fbSdoErrorFieldValue[6]);		
END_IF

// Check for error field 7
IF Status.nNumErrors >= 7 THEN
	fbSdoErrorField_7(bStartReading := TRUE);
	IF fbSdoErrorField_7.ReadDataAvailable THEN
		fbSdoErrorFieldValue[7] := fbSdoErrorField_7.GetReadDataAsUDINT();
		Status.ErrorField[7] := ParseErrorField(fbSdoErrorFieldValue[7]);
	END_IF
ELSE
	fbSdoErrorFieldValue[7] := 0;
	Status.ErrorField[7] := ParseErrorField(fbSdoErrorFieldValue[7]);		
END_IF

// Check for error field 8
IF Status.nNumErrors >= 8 THEN
	fbSdoErrorField_8(bStartReading := TRUE);
	IF fbSdoErrorField_8.ReadDataAvailable THEN
		fbSdoErrorFieldValue[8] := fbSdoErrorField_8.GetReadDataAsUDINT();
		Status.ErrorField[8] := ParseErrorField(fbSdoErrorFieldValue[8]);
	END_IF
ELSE
	fbSdoErrorFieldValue[8] := 0;
	Status.ErrorField[8] := ParseErrorField(fbSdoErrorFieldValue[8]);		
END_IF
END_ACTION

METHOD PUBLIC CheckModesOfOperation : BOOL
VAR_INPUT
END_VAR
CASE stPDOs.TxPDO_1_6061h_ModesOfOperationDisplay OF
	
	-2:
		eModesOfOperation := E_PDxx_ModesOfOperation.AUTO_SETUP;
	-1:
		eModesOfOperation := E_PDxx_ModesOfOperation.CLOCK_DIRECTION_MODE;
	0:
		eModesOfOperation := E_PDxx_ModesOfOperation.NO_MODE_CHANGE_OR_NO_MODE_ASSIGNED;
	1:
		eModesOfOperation := E_PDxx_ModesOfOperation.PROFILE_POSITION_MODE;
	2:
		eModesOfOperation := E_PDxx_ModesOfOperation.VELOCITY_MODE;
	3:
		eModesOfOperation := E_PDxx_ModesOfOperation.PROFILE_VELOCITY_MODE;
	4:
		eModesOfOperation := E_PDxx_ModesOfOperation.PROFILE_TORQUE_MODE;
	5:
		eModesOfOperation := E_PDxx_ModesOfOperation.RESERVED;
	6:
		eModesOfOperation := E_PDxx_ModesOfOperation.HOMING_MODE;
	7:
		eModesOfOperation := E_PDxx_ModesOfOperation.INTERPOLATED_POSITION_MODE;
	8:
		eModesOfOperation := E_PDxx_ModesOfOperation.CYCLIC_SYNCHRONOUS_POSITION_MODE;
	9:
		eModesOfOperation := E_PDxx_ModesOfOperation.CYCLIC_SYNCHRONOUS_VELOCITY_MODE;
	10:
		eModesOfOperation := E_PDxx_ModesOfOperation.CYCLIC_SYNCHRONOUS_TORQUE_MODE;	

END_CASE
END_METHOD

METHOD PUBLIC CheckState
(* Following comments are from PD2-C manual, section "6041h Statusword" on p. 279-280 *)
VAR
	LowerNibble : BYTE; // 4 bit container to hold the combination of RTSO, SO, OE and FAULT bits. Highest 4 bit in the BYTE should always be zero.
END_VAR
stStatusWord.ReadyToSwitchOn				:= stPDOs.TxPDO_1_6041h_StatusWord.0;
stStatusWord.SwitchedOn						:= stPDOs.TxPDO_1_6041h_StatusWord.1;
stStatusWord.OperationEnabled				:= stPDOs.TxPDO_1_6041h_StatusWord.2;
stStatusWord.Fault							:= stPDOs.TxPDO_1_6041h_StatusWord.3;
stStatusWord.VoltageEnabled					:= stPDOs.TxPDO_1_6041h_StatusWord.4;
stStatusWord.QuickStop						:= stPDOs.TxPDO_1_6041h_StatusWord.5;
stStatusWord.SwitchOnDisabled				:= stPDOs.TxPDO_1_6041h_StatusWord.6;
stStatusWord.Warning						:= stPDOs.TxPDO_1_6041h_StatusWord.7;
stStatusWord.Synchronization				:= stPDOs.TxPDO_1_6041h_StatusWord.8;
stStatusWord.Remote							:= stPDOs.TxPDO_1_6041h_StatusWord.9;
stStatusWord.TargetReached 					:= stPDOs.TxPDO_1_6041h_StatusWord.10;
stStatusWord.InternalLimitReached			:= stPDOs.TxPDO_1_6041h_StatusWord.11;
stStatusWord.OperationModeSpecific_bit12	:= stPDOs.TxPDO_1_6041h_StatusWord.12;
stStatusWord.OperationModeSpecific_bit13	:= stPDOs.TxPDO_1_6041h_StatusWord.13;
stStatusWord.ClosedLoopAvailable			:= stPDOs.TxPDO_1_6041h_StatusWord.15;

LowerNibble 	:= 0;
LowerNibble.0	:= stPDOs.TxPDO_1_6041h_StatusWord.0;
LowerNibble.1	:= stPDOs.TxPDO_1_6041h_StatusWord.1;
LowerNibble.2	:= stPDOs.TxPDO_1_6041h_StatusWord.2;
LowerNibble.3	:= stPDOs.TxPDO_1_6041h_StatusWord.3;

(* Listed in the following table are the bit masks that break down the state of the controller
xxxx xxxx x0xx 0000 Not ready to switch on
xxxx xxxx x1xx 0000 Switch on disabled
xxxx xxxx x01x 0001 Ready to switch on
xxxx xxxx x01x 0011 Switched on
xxxx xxxx x01x 0111 Operation enabled
xxxx xxxx x00x 0111 Quick stop active
xxxx xxxx x0xx 1111 Fault reaction active
xxxx xxxx x0xx 1000 Fault
*)

IF 		NOT stStatusWord.SwitchOnDisabled 									AND LowerNibble = 2#0000 THEN 	eState := E_PDxx_State.NOT_READY_TO_SWITCH_ON;
ELSIF  		stStatusWord.SwitchOnDisabled 									AND LowerNibble = 2#0000 THEN	eState := E_PDxx_State.SWITCH_ON_DISABLED;
ELSIF 	NOT stStatusWord.SwitchOnDisabled AND 		stStatusWord.QuickStop 	AND LowerNibble = 2#0001 THEN	eState := E_PDxx_State.READY_TO_SWITCH_ON;
ELSIF 	NOT stStatusWord.SwitchOnDisabled AND 		stStatusWord.QuickStop 	AND LowerNibble = 2#0011 THEN	eState := E_PDxx_State.SWITCHED_ON;
ELSIF 	NOT stStatusWord.SwitchOnDisabled AND 		stStatusWord.QuickStop	AND LowerNibble = 2#0111 THEN	eState := E_PDxx_State.OPERATION_ENABLED;
ELSIF 	NOT stStatusWord.SwitchOnDisabled AND NOT 	stStatusWord.QuickStop 	AND LowerNibble = 2#0111 THEN	eState := E_PDxx_State.QUICK_STOP_ACTIVE;
ELSIF 	NOT stStatusWord.SwitchOnDisabled									AND LowerNibble = 2#1111 THEN	eState := E_PDxx_State.FAULT_REACTION_ACTIVE;
ELSIF 	NOT stStatusWord.SwitchOnDisabled									AND LowerNibble = 2#1000 THEN	eState := E_PDxx_State.FAULT;
ELSE																										eState := E_PDxx_State.UNKNOWN_STATE;	
END_IF

IF eState = E_PDxx_State.FAULT THEN
	ChangeState(E_PDxx_State.SWITCH_ON_DISABLED);
END_IF

Status.nCurrentPosition := GetPosition();
Status.nCurrentVelocity := GetVelocity();
END_METHOD


METHOD PUBLIC ClearErrorFields : BOOL

fbSdoNumberOfErrors.SetWriteDataFromUSINT(0);
fbSdoNumberOfErrors(bStartWriting := TRUE);

ClearErrorFields := Status.nNumErrors = 0;
END_METHOD

METHOD PUBLIC EnableOperation : BOOL
CASE eState OF
	E_PDxx_State.SWITCH_ON_DISABLED:
		ChangeState(E_PDxx_State.READY_TO_SWITCH_ON);
		ChangeModesOfOperation(E_PDxx_ModesOfOperation.PROFILE_POSITION_MODE);				
	E_PDxx_State.READY_TO_SWITCH_ON:
		ChangeState(E_PDxx_State.SWITCHED_ON);
	E_PDxx_State.SWITCHED_ON:
		ChangeState(E_PDxx_State.OPERATION_ENABLED);
END_CASE

IF eState = E_PDxx_State.OPERATION_ENABLED AND 
eModesOfOperation = E_PDxx_ModesOfOperation.PROFILE_POSITION_MODE THEN
	EnableOperation := TRUE;
ELSE
	EnableOperation := FALSE;
END_IF
END_METHOD

METHOD PUBLIC GetActualPosition : DINT
GetActualPosition := stPDOs.TxPDO_2_6064h_PositionActualValue;
END_METHOD

METHOD PRIVATE GetActualPositionFromNormalisedPosition : DINT
VAR_INPUT
	nNormalisedPosition : DINT;
END_VAR
IF Status.bReversePolarity = TRUE THEN
	GetActualPositionFromNormalisedPosition := Status.nMaxActualPosition - nNormalisedPosition;
ELSE
	GetActualPositionFromNormalisedPosition := nNormalisedPosition + Status.nMinActualPosition;	
END_IF
END_METHOD

METHOD PUBLIC GetCurrent : UDINT
GetCurrent := fbSdoMaxCurrentValue;
END_METHOD

METHOD PUBLIC GetDigitalInputs
VAR_OUTPUT
	stDigitalInputs : ST_PDxx_IO;
END_VAR
stDigitalInputs := stIO;
END_METHOD

METHOD PRIVATE GetNormalisedPositionFromActualPosition : DINT
VAR_INPUT
	nActualPosition : DINT;
END_VAR
IF Status.bReversePolarity = TRUE THEN
	GetNormalisedPositionFromActualPosition := Status.nMaxActualPosition - nActualPosition;
ELSE
	GetNormalisedPositionFromActualPosition := nActualPosition - Status.nMinActualPosition;	
END_IF
END_METHOD

METHOD PUBLIC GetPosition : DINT
GetPosition := GetNormalisedPositionFromActualPosition(stPDOs.TxPDO_2_6064h_PositionActualValue);
END_METHOD

METHOD PUBLIC GetVelocity : INT
IF Status.bReversePolarity = TRUE THEN
//	 GetVelocity := -stPDOs.RxPDO_3_6042h_TargetVelocity;
	 GetVelocity := -stPDOs.TxPDO_3_6044h_VelocityActualValue;
ELSE
//	GetVelocity := stPDOs.RxPDO_3_6042h_TargetVelocity;	
	GetVelocity := stPDOs.TxPDO_3_6044h_VelocityActualValue;	
END_IF
END_METHOD

METHOD PUBLIC GoToTargetPosition : DINT
VAR_INPUT
	nPosition 	: DINT;
	nVelocity	: INT;
	nMaxCurrent	: UDINT;
END_VAR
VAR_INST
	diff 		: DINT;
	startMoveInCycles : ULINT := 0;
END_VAR
diff := GetPosition() - nPosition;

IF fbSdoMaxCurrentValue <> nMaxCurrent THEN
	SetMaxCurrent(nMaxCurrent);
ELSE
	SetProfileVelocity(nVelocity);
	IF SetProfilePositionMode() = TRUE THEN
		IF SetTargetPosition(nRequestedPosition := nPosition) = TRUE THEN
			startMoveInCycles := 2;
		END_IF
		IF startMoveInCycles = 1 THEN
			StartMoveToTargetPosition();
			startMoveInCycles := 0;
		ELSIF startMoveInCycles > 0 THEN
			startMoveInCycles := startMoveInCycles - 1;
		END_IF
	END_IF
END_IF

GoToTargetPosition := diff;
END_METHOD


METHOD PUBLIC GoToTargetVelocity : INT
VAR_INPUT
	nVelocity	: INT;
	nMaxCurrent	: UDINT;
END_VAR
IF fbSdoMaxCurrentValue <> nMaxCurrent THEN
	SetMaxCurrent(nMaxCurrent);
ELSE
	IF SetVelocityMode() THEN
		SetTargetVelocity(-nVelocity); // It is negative because we want to move towards the closed position zero point from a positive valued open gripper.
	END_IF	
END_IF

GoToTargetVelocity := nVelocity - GetVelocity();
END_METHOD

METHOD PUBLIC GripThickness : DINT
VAR_INPUT
	nObjectThickness 	: DINT;
	nVelocity			: INT;
	nMaxCurrent			: UDINT;
END_VAR
IF fbSdoMaxCurrentValue <> nMaxCurrent THEN
	SetMaxCurrent(nMaxCurrent);
ELSE
	IF SetVelocityMode() THEN
		SetTargetVelocity(-nVelocity); // It is negative because we want to move towards the closed position zero point from a positive valued open gripper.
		Status.nTargetPosition := GetPosition();
	END_IF	
END_IF

GripThickness := GetPosition() - nObjectThickness;
END_METHOD

METHOD PUBLIC IsPolarityReversed : BOOL
IsPolarityReversed := Status.bReversePolarity;
END_METHOD


METHOD ParseErrorField : ST_PDxx_PredefinedErrorField
VAR_INPUT
	nErrorFieldAsUDINT : UDINT;
END_VAR

ParseErrorField.nErrorCode 		:= UDINT_TO_UINT(nErrorFieldAsUDINT);
ParseErrorField.stErrorClass	:= ParseErrorRegister(UDINT_TO_USINT(SHR(nErrorFieldAsUDINT,16)));
ParseErrorField.nErrorNumber	:= UDINT_TO_USINT(SHR(nErrorFieldAsUDINT,24));
END_METHOD


METHOD PUBLIC ParseErrorRegister : ST_PDxx_ErrorRegister
VAR_INPUT
	nErrorRegisterAsUSINT : USINT;
END_VAR

ParseErrorRegister.GEN 	:= nErrorRegisterAsUSINT.0; // General Error
ParseErrorRegister.CUR 	:= nErrorRegisterAsUSINT.1; // Current
ParseErrorRegister.VOL 	:= nErrorRegisterAsUSINT.2; // Voltage
ParseErrorRegister.TEMP := nErrorRegisterAsUSINT.3; // Temperature
ParseErrorRegister.COM	:= nErrorRegisterAsUSINT.4; // Communication
ParseErrorRegister.PROF	:= nErrorRegisterAsUSINT.5; // Relates to the device profile
ParseErrorRegister.RES	:= nErrorRegisterAsUSINT.6; // Reserved, always "0"
ParseErrorRegister.MAN	:= nErrorRegisterAsUSINT.7; // Manufacturer-specific : The motor turns in the wrong direction
END_METHOD


METHOD PUBLIC ProbeActualPositionLimits : BOOL
VAR_INPUT
	nVelocity : INT;
END_VAR

VAR_INST
	nMinStartActualPosition : DINT;
	nMaxStartActualPosition : DINT;
END_VAR

VAR
	nActualVelocity			: INT;
	nActualPosition			: DINT;
END_VAR

(* 	Returns true whenever the method was able to push past
	one of the limits. External function can monitor how 
	long this method has returned FALSE, in order to 
	determine whether a end limit has been found. *)

IF SetVelocityMode() THEN
	SetTargetVelocity(nVelocity);
ELSE
	Status.nMaxActualPosition := GetActualPosition();
	Status.nMinActualPosition := GetActualPosition();
	nMaxStartActualPosition := Status.nMaxActualPosition;
	nMinStartActualPosition := Status.nMinActualPosition;
	ProbeActualPositionLimits := TRUE;
END_IF

//IF IsPolarityReversed() = TRUE THEN
IF Status.bReversePolarity = TRUE THEN
	nActualVelocity := -nVelocity;
ELSE
	nActualVelocity := nVelocity;
END_IF

nActualPosition := GetActualPosition();

IF nActualVelocity > 0 AND nActualPosition > Status.nMaxActualPosition THEN
	Status.nMaxActualPosition := nActualPosition;
	ProbeActualPositionLimits := TRUE;
ELSIF nActualVelocity < 0 AND nActualPosition < Status.nMinActualPosition THEN
	Status.nMinActualPosition := nActualPosition;
	ProbeActualPositionLimits := TRUE;
ELSE
	IF (nActualVelocity > 0 AND nActualPosition > nMaxStartActualPosition) OR
	   (nActualVelocity < 0 AND nActualPosition < nMinStartActualPosition) THEN
		ProbeActualPositionLimits := FALSE;
	ELSE
		ProbeActualPositionLimits := TRUE;
	END_IF
END_IF

Status.nTargetPosition := GetPosition();
END_METHOD

METHOD PUBLIC ReleaseGripToThicknessMargin : DINT
VAR_INPUT
	nObjectThickness 		: DINT;
	nObjectReleaseMargin	: DINT;
	nVelocity				: INT;
	nMaxCurrent				: UDINT;
END_VAR
ReleaseGripToThicknessMargin := GoToTargetPosition(	nPosition 	:= nObjectThickness + nObjectReleaseMargin,
													nVelocity 	:= nVelocity,
													nMaxCurrent	:= nMaxCurrent);
END_METHOD


METHOD PRIVATE ResetControlWordBit4 : BOOL
VAR_INPUT
END_VAR

IF eState = E_PDxx_State.OPERATION_ENABLED AND 
   eModesOfOperation = E_PDxx_ModesOfOperation.PROFILE_POSITION_MODE AND
   stControlWord.OperationModeSpecific_bit_4 = TRUE AND
   stStatusWord.OperationModeSpecific_bit12 = TRUE THEN
	stControlWord.OperationModeSpecific_bit_4 := FALSE;
	stPDOs.RxPDO_1_6040h_ControlWord.4 := stControlWord.OperationModeSpecific_bit_4;	
END_IF
END_METHOD

ACTION ResetStatusAndSDOs:

Status.bZeroInitialised		:= FALSE;
Status.bReversePolarity		:= FALSE;
Status.nHomePosition 		:= 0;
Status.nCurrentPosition		:= 0;
Status.nCurrentVelocity		:= 0;
Status.nTargetPosition		:= 0;
Status.nMinActualPosition	:= 0;
Status.nMaxActualPosition	:= 0;

fbSdoMaxCurrentValue 			:= 0;
fbSdoSpecialFunctionEnableValue	:= 0;
fbSdoFunctionInvertedValue		:= 0;
fbSdoInputRangeSelectValue		:= 0;
fbSdoFeedValue					:= 0;
fbSdoShaftRevolutionsValue		:= 0;
fbSdoEncoderIncrementsValue		:= 0;
fbSdoMotorRevolutionsValue		:= 0;
fbSdoSIUnitPositionValue		:= 0;
END_ACTION

METHOD PUBLIC SetFeedRate : BOOL
VAR_INPUT
	nFeedRate				: UDINT;
	nDivisor				: UDINT;
END_VAR
VAR
	nFeed					: UDINT;
	nShaftRevolutions		: UDINT;
END_VAR
VAR_INST
	bEncoderIncrementsRead	: BOOL := FALSE;
	bMotorRevolutionsRead	: BOOL := FALSE;
END_VAR

fbSdoEncoderIncrements(bStartReading := TRUE);
IF fbSdoEncoderIncrements.ReadDataAvailable THEN
	fbSdoEncoderIncrementsValue := fbSdoEncoderIncrements.GetReadDataAsUDINT();
	bEncoderIncrementsRead := TRUE;
END_IF

fbSdoMotorRevolutions(bStartReading := TRUE);
IF fbSdoMotorRevolutions.ReadDataAvailable THEN
	fbSdoMotorRevolutionsValue := fbSdoMotorRevolutions.GetReadDataAsUDINT();
	bMotorRevolutionsRead := TRUE;
END_IF

IF bEncoderIncrementsRead AND bMotorRevolutionsRead THEN
	nFeed := nFeedRate;// * fbSdoMotorRevolutionsValue; // commented out part was clashing with SetSIUnitPosition on PD4-E
	nShaftRevolutions := nDivisor;// * fbSdoEncoderIncrementsValue;  // commented out part was clashing with SetSIUnitPosition on PD4-E
  
	fbSdoFeed.SetWriteDataFromUDINT(nFeed);
	fbSdoFeed(bStartReading := TRUE);
	
	IF fbSdoFeed.ReadDataAvailable THEN
		fbSdoFeedValue := fbSdoFeed.GetReadDataAsUDINT();
	END_IF
	
	IF fbSdoFeedValue <> nFeed THEN
		fbSdoFeed(bStartWriting := TRUE);
	END_IF
	
	fbSdoShaftRevolutions.SetWriteDataFromUDINT(nShaftRevolutions);
	fbSdoShaftRevolutions(bStartReading := TRUE, bStartWriting := TRUE);
	
	IF fbSdoShaftRevolutions.ReadDataAvailable THEN
		fbSdoShaftRevolutionsValue := fbSdoShaftRevolutions.GetReadDataAsUDINT();
	END_IF
	
	IF fbSdoShaftRevolutionsValue <> nShaftRevolutions THEN
		fbSdoShaftRevolutions(bStartWriting := TRUE);
	END_IF
	
	IF fbSdoFeedValue = nFeed AND
		fbSdoShaftRevolutionsValue = nShaftRevolutions THEN
		SetFeedRate := TRUE;
	ELSE
		SetFeedRate := FALSE;
	END_IF
END_IF

//fbSdoFeed.SetWriteDataFromUDINT(nFeed);
//fbSdoFeed(bStartReading := TRUE);

//IF fbSdoFeed.ReadDataAvailable THEN
//	fbSdoFeedValue := fbSdoFeed.GetReadDataAsUDINT();
//END_IF

//IF fbSdoFeedValue <> nFeedRate THEN
//	fbSdoFeed(bStartWriting := TRUE);
//END_IF

//fbSdoShaftRevolutions.SetWriteDataFromUDINT(nShaftRevolutions);
//fbSdoShaftRevolutions(bStartReading := TRUE, bStartWriting := TRUE);

//IF fbSdoShaftRevolutions.ReadDataAvailable THEN
//	fbSdoShaftRevolutionsValue := fbSdoShaftRevolutions.GetReadDataAsUDINT();
//END_IF

//IF fbSdoShaftRevolutionsValue <> nShaftRevolutions THEN
//	fbSdoShaftRevolutions(bStartWriting := TRUE);
//END_IF

//IF fbSdoFeedValue = nFeedRate AND
//	fbSdoShaftRevolutionsValue = nShaftRevolutions THEN
//	SetFeedRate := TRUE;
//ELSE
//	SetFeedRate := FALSE;
//END_IF
END_METHOD

METHOD PUBLIC SetHomePosition
VAR_INPUT
	nPosition : DINT;
END_VAR
Status.nHomePosition := nPosition;
END_METHOD

METHOD PUBLIC SetMaxCurrent : BOOL
VAR_INPUT
	nMaxCurrent : UDINT;
END_VAR
fbSdoMaxCurrent.SetWriteDataFromUDINT(nMaxCurrent);
fbSdoMaxCurrent(bStartReading := TRUE, bStartWriting := TRUE);

IF SimParameters.bActivateSimulation = TRUE THEN
	fbSdoMaxCurrentValue := nMaxCurrent;
ELSE
	IF fbSdoMaxCurrent.ReadDataAvailable THEN
		fbSdoMaxCurrentValue := fbSdoMaxCurrent.GetReadDataAsUDINT();
	END_IF
END_IF
		
IF fbSdoMaxCurrentValue = nMaxCurrent THEN
	SetMaxCurrent := TRUE;
ELSE
	SetMaxCurrent := FALSE;
END_IF
END_METHOD


METHOD PUBLIC SetProfileAcceleration : BOOL
VAR_INPUT
	nProfileAcceleration : UDINT;
END_VAR

fbSdoProfileAcceleration.SetWriteDataFromUDINT(nProfileAcceleration);
fbSdoProfileAcceleration(bStartReading := TRUE, bStartWriting := TRUE);

IF SimParameters.bActivateSimulation = TRUE THEN
	fbSdoProfileAccelerationValue := nProfileAcceleration;
ELSE
	IF fbSdoProfileAcceleration.ReadDataAvailable THEN
		fbSdoProfileAccelerationValue := fbSdoProfileAcceleration.GetReadDataAsUDINT();
	END_IF
END_IF
		
IF fbSdoProfileAccelerationValue = nProfileAcceleration THEN
	SetProfileAcceleration := TRUE;
ELSE
	SetProfileAcceleration := FALSE;
END_IF
END_METHOD


METHOD PUBLIC SetProfileDeceleration : BOOL
VAR_INPUT
	nProfileDeceleration : UDINT;
END_VAR

fbSdoProfileDeceleration.SetWriteDataFromUDINT(nProfileDeceleration);
fbSdoProfileDeceleration(bStartReading := TRUE, bStartWriting := TRUE);

IF SimParameters.bActivateSimulation = TRUE THEN
	fbSdoProfileDecelerationValue := nProfileDeceleration;
ELSE
	IF fbSdoProfileDeceleration.ReadDataAvailable THEN
		fbSdoProfileDecelerationValue := fbSdoProfileDeceleration.GetReadDataAsUDINT();
	END_IF
END_IF
		
IF fbSdoProfileDecelerationValue = nProfileDeceleration THEN
	SetProfileDeceleration := TRUE;
ELSE
	SetProfileDeceleration := FALSE;
END_IF
END_METHOD

METHOD PUBLIC SetProfilePositionMode : BOOL
CASE eState OF
	E_PDxx_State.SWITCH_ON_DISABLED,
	E_PDxx_State.READY_TO_SWITCH_ON:
		SwitchOnPowerToMotor();
	E_PDxx_State.SWITCHED_ON:
		IF eModesOfOperation <> E_PDxx_ModesOfOperation.PROFILE_POSITION_MODE THEN
			ChangeModesOfOperation(E_PDxx_ModesOfOperation.PROFILE_POSITION_MODE);
		ELSE
			ChangeState(E_PDxx_State.OPERATION_ENABLED);
		END_IF	
	E_PDxx_State.OPERATION_ENABLED:
		IF eModesOfOperation <> E_PDxx_ModesOfOperation.PROFILE_POSITION_MODE THEN
			ChangeState(E_PDxx_State.SWITCHED_ON);			
		END_IF
END_CASE

IF eState = E_PDxx_State.OPERATION_ENABLED AND 
eModesOfOperation = E_PDxx_ModesOfOperation.PROFILE_POSITION_MODE THEN
	SetProfilePositionMode := TRUE;
ELSE
	SetProfilePositionMode := FALSE;
END_IF
END_METHOD


METHOD PUBLIC SetProfileVelocity
VAR_INPUT
	nVelocity : INT;
END_VAR

IF nVelocity < 0 THEN
	stPDOs.RxPDO_2_6081h_ProfileVelocity := INT_TO_UDINT(-nVelocity);
ELSE
	stPDOs.RxPDO_2_6081h_ProfileVelocity := INT_TO_UDINT(nVelocity);	
END_IF
END_METHOD

METHOD PUBLIC SetRangeForDigitalInput : BOOL
VAR_INPUT
	nInputNumber	: USINT;
	bEnable24V		: BOOL;
END_VAR

VAR
	bReadValue		: BOOL;
END_VAR
fbSdoInputRangeSelect(bStartReading := TRUE);

IF fbSdoInputRangeSelect.ReadDataAvailable THEN
	fbSdoInputRangeSelectValue := fbSdoInputRangeSelect.GetReadDataAsUDINT();
	CASE nInputNumber OF
		1:
			bReadValue := fbSdoInputRangeSelectValue.0;
		2:
			bReadValue := fbSdoInputRangeSelectValue.1;
		3:
			bReadValue := fbSdoInputRangeSelectValue.2;
		4:
			bReadValue := fbSdoInputRangeSelectValue.3;
	END_CASE
	IF bReadValue <> bEnable24V THEN
		CASE nInputNumber OF
			1:
				stIO.Input1_24V := bEnable24V;
			2:
				stIO.Input2_24V := bEnable24V;
			3:
				stIO.Input3_24V := bEnable24V;
			4:
				stIO.Input4_24V := bEnable24V;
		END_CASE
		fbSdoInputRangeSelectValue.0 := stIO.Input1_24V;
		fbSdoInputRangeSelectValue.1 := stIO.Input2_24V;
		fbSdoInputRangeSelectValue.2 := stIO.Input3_24V;
		fbSdoInputRangeSelectValue.3 := stIO.Input4_24V;
		fbSdoInputRangeSelectValue.4 := stIO.Input5_24V;
		fbSdoInputRangeSelectValue.5 := stIO.Input6_24V;
		fbSdoInputRangeSelectValue.6 := stIO.Input7_24V;
		fbSdoInputRangeSelectValue.7 := stIO.Input8_24V;
		
		fbSdoInputRangeSelect(bStartReading := TRUE, bStartWriting := TRUE);
		SetRangeForDigitalInput := FALSE;
	ELSE
		SetRangeForDigitalInput := TRUE;	
	END_IF
ELSE
	SetRangeForDigitalInput := FALSE;
END_IF
END_METHOD

METHOD PUBLIC SetReversePolarity : BOOL
VAR_INPUT
	bReversePositionAndVelocity : BOOL;
END_VAR
IF stStatusWord.OperationEnabled THEN
	SetReversePolarity := FALSE;
ELSE
	Status.bReversePolarity := bReversePositionAndVelocity;
	SetReversePolarity := TRUE;	
END_IF
END_METHOD

METHOD PUBLIC SetSIUnitPosition : BOOL
VAR_INPUT
	nUnit					: USINT;
	nFactor					: USINT;
END_VAR
VAR
	nSIUnitPosition			: UDINT;
//	bSIUnitPositionRead		: BOOL;
END_VAR
nSIUnitPosition := nFactor;
nSIUnitPosition := SHL(nSIUnitPosition, 8);
nSIUnitPosition := nSIUnitPosition + nUnit;
nSIUnitPosition := SHL(nSIUnitPosition, 16);

fbSdoSIUnitPosition.SetWriteDataFromUDINT(nSIUnitPosition);
fbSdoSIUnitPosition(bStartReading := TRUE, bStartWriting := TRUE);

IF fbSdoSIUnitPosition.ReadDataAvailable THEN
	fbSdoSIUnitPositionValue := fbSdoSIUnitPosition.GetReadDataAsUDINT();
//	bSIUnitPositionRead := TRUE;
END_IF
	
IF fbSdoSIUnitPositionValue = nSIUnitPosition THEN
	SetSIUnitPosition := TRUE;
ELSE
	SetSIUnitPosition := FALSE;
END_IF
END_METHOD


METHOD PRIVATE SetTargetPosition : BOOL
VAR_INPUT
	nRequestedPosition : DINT;
END_VAR

IF Status.nTargetPosition <> nRequestedPosition AND
   stStatusWord.OperationModeSpecific_bit12 = FALSE AND
   stControlWord.OperationModeSpecific_bit_4 = FALSE THEN
	Status.nTargetPosition := nRequestedPosition;
	stPDOs.RxPDO_2_607Ah_TargetPosition := GetActualPositionFromNormalisedPosition(Status.nTargetPosition);
	SetTargetPosition := TRUE;
ELSE
	SetTargetPosition := FALSE;
END_IF
END_METHOD

METHOD PUBLIC SetTargetVelocity
VAR_INPUT
	nVelocity : INT;
END_VAR
IF Status.bReversePolarity = TRUE THEN
	stPDOs.RxPDO_3_6042h_TargetVelocity := -nVelocity;;
ELSE
	stPDOs.RxPDO_3_6042h_TargetVelocity := nVelocity;;	
END_IF
END_METHOD

METHOD PUBLIC SetVelocityMode : BOOL
VAR_INPUT
END_VAR
CASE eState OF
	E_PDxx_State.SWITCH_ON_DISABLED,
	E_PDxx_State.READY_TO_SWITCH_ON:
		SwitchOnPowerToMotor();
	E_PDxx_State.SWITCHED_ON:
		SetTargetVelocity(0);
		IF eModesOfOperation <> E_PDxx_ModesOfOperation.VELOCITY_MODE THEN
			ChangeModesOfOperation(E_PDxx_ModesOfOperation.VELOCITY_MODE);
		ELSE
			ChangeState(E_PDxx_State.OPERATION_ENABLED);
		END_IF
	E_PDxx_State.OPERATION_ENABLED:
		IF eModesOfOperation <> E_PDxx_ModesOfOperation.VELOCITY_MODE THEN
			ChangeState(E_PDxx_State.SWITCHED_ON);			
		END_IF
END_CASE

IF eState = E_PDxx_State.OPERATION_ENABLED AND 
eModesOfOperation = E_PDxx_ModesOfOperation.VELOCITY_MODE THEN
	SetVelocityMode := TRUE;
ELSE
	SetVelocityMode := FALSE;
END_IF
END_METHOD

METHOD PUBLIC SetZeroPositionHere
IF Status.bReversePolarity = TRUE THEN
	Status.nMaxActualPosition := GetActualPosition();
ELSE
	Status.nMinActualPosition := GetActualPosition();
END_IF
END_METHOD

METHOD PRIVATE StartMoveToTargetPosition : BOOL

VAR
	ControlWord : UINT;
END_VAR
IF 	SetProfilePositionMode() THEN
	
	stControlWord.SwitchedOn_bit_0				:= TRUE;
	stControlWord.EnableVoltage_bit_1			:= TRUE;
	stControlWord.QuickStop_bit_2				:= TRUE; // Quick stop is Active Low
	stControlWord.EnableOperation_bit_3			:= TRUE;
	stControlWord.FaultReset_bit_7				:= FALSE;
	stControlWord.OperationModeSpecific_bit_4	:= TRUE;
	stControlWord.OperationModeSpecific_bit_5	:= FALSE;
	stControlWord.OperationModeSpecific_bit_6	:= FALSE;
	stControlWord.Halt_bit_8					:= FALSE;
	stControlWord.OperationModeSpecific_bit_9	:= FALSE;
	
	ControlWord.0 := stControlWord.SwitchedOn_bit_0;
	ControlWord.1 := stControlWord.EnableVoltage_bit_1;
	ControlWord.2 := stControlWord.QuickStop_bit_2;
	ControlWord.3 := stControlWord.EnableOperation_bit_3;
	ControlWord.4 := stControlWord.OperationModeSpecific_bit_4;
	ControlWord.5 := stControlWord.OperationModeSpecific_bit_5;
	ControlWord.6 := stControlWord.OperationModeSpecific_bit_6;
	ControlWord.7 := stControlWord.FaultReset_bit_7;
	ControlWord.8 := stControlWord.Halt_bit_8;
	ControlWord.9 := stControlWord.OperationModeSpecific_bit_9;
	
	stPDOs.RxPDO_1_6040h_ControlWord := ControlWord;
	StartMoveToTargetPosition := TRUE;
ELSE
	StartMoveToTargetPosition := FALSE;
END_IF
END_METHOD

METHOD PUBLIC SwitchOffPowerToMotor : BOOL
CASE eState OF
	E_PDxx_State.READY_TO_SWITCH_ON,
	E_PDxx_State.SWITCHED_ON,	
	E_PDxx_State.OPERATION_ENABLED:
		ChangeState(E_PDxx_State.SWITCH_ON_DISABLED);
END_CASE

IF eState = E_PDxx_State.SWITCH_ON_DISABLED THEN
	SwitchOffPowerToMotor := TRUE;
	Status.nTargetPosition := GetPosition();
ELSE
	SwitchOffPowerToMotor := FALSE;
END_IF
END_METHOD

METHOD PUBLIC SwitchOnPowerToMotor : BOOL
CASE eState OF
	E_PDxx_State.SWITCH_ON_DISABLED:
		ChangeState(E_PDxx_State.READY_TO_SWITCH_ON);
	E_PDxx_State.READY_TO_SWITCH_ON:
		ChangeState(E_PDxx_State.SWITCHED_ON);
END_CASE

IF eState = E_PDxx_State.SWITCHED_ON THEN
	SwitchOnPowerToMotor := TRUE;
	Status.nTargetPosition := GetPosition();
ELSE
	SwitchOnPowerToMotor := FALSE;
END_IF
END_METHOD

END_FUNCTION_BLOCK

// ---- POUs/FB_SDO.TcPOU
FUNCTION_BLOCK FB_SDO
VAR_INPUT
	bStartReading	: BOOL;		(* only reset to FALSE after ReadDataAvailable=TRUE*)
	bStartWriting	: BOOL;		(* only reset to FALSE after WriteDataFinished=TRUE*)
END_VAR
VAR
	CO_Name			: STRING[255] := 'UNNAMED CANopen Object';
	CO_Index		: DWORD;	(* This is the Index of the CANopen Object Dictionary Entry*)
	CO_SubIndex		: DWORD;	(* This is the Sub-Index of the CANopen Object Dictionary Entry*)
	DataLength		: DWORD;	(* This is the Length of the CANopen Object Dictionary Entry*)
	stCANopenDevice	: REFERENCE TO ST_CANopenDevice;
	ReadData		: ARRAY[0..255] OF BYTE;
    WriteData		: ARRAY[0..255] OF BYTE; (* This array contains the data to be written to the CANopen Object Dictionary*)
    ReadDataAvailable:BOOL;
	WriteDataFinished:BOOL;
    Error			: DWORD;
    ReadState		: BYTE := 0;
	WriteState		: BYTE := 0;
    ADSRead 		: ADSREAD;
	ADSWrite		: ADSWRITE;

END_VAR

CASE ReadState OF
    0:
        IF bStartReading THEN
           ReadDataAvailable := FALSE;
           Error := 0;
           ADSRead(
               NETID:= stCANopenDevice.AmsNetId,
               PORT:= stCANopenDevice.PortNr,
               IDXGRP:= CO_Index,
               IDXOFFS:= CO_SubIndex,
               LEN:= DataLength,
               DESTADDR:= ADR(ReadData),
               READ:= TRUE,
               TMOUT := T#1s
               );
           IF ADSRead.err THEN
               ReadState := 2;
               ReadDataAvailable := TRUE;
               Error := ADSRead.ErrId;
           ELSE
               ReadState := 1;
           END_IF
        ELSE
           ADSRead(
               NETID:= stCANopenDevice.AmsNetId,
               PORT:= stCANopenDevice.PortNr,
               IDXGRP:= CO_Index,
               IDXOFFS:= CO_SubIndex,
               LEN:= DataLength,
               DESTADDR:= ADR(ReadData),
               READ:= FALSE,
               TMOUT := T#1s
           );
        END_IF
    1:
        ADSRead(READ:= FALSE);
        IF ADSRead.err THEN
           ReadState := 2;
           ReadDataAvailable := TRUE;
           Error := ADSRead.ErrId;
        ELSE
           IF NOT ADSRead.busy THEN
               ReadState := 2;
               ReadDataAvailable := TRUE;
           END_IF
        END_IF
    2:
        ADSRead(READ:= FALSE);
		bStartReading := FALSE;
        ReadState := 0;
END_CASE

CASE
WriteState OF
    0:
        IF bStartWriting THEN
           WriteDataFinished := FALSE;
           Error := 0;
           ADSWrite(
               NETID:= stCANopenDevice.AmsNetId,
               PORT:= stCANopenDevice.PortNr,
               IDXGRP:= CO_Index,
               IDXOFFS:= CO_SubIndex,
               LEN:= DataLength,
               SRCADDR:= ADR(WriteData),
               WRITE:= TRUE,
               TMOUT := T#1s
               );
           IF ADSWrite.err THEN
               WriteState := 2;
               WriteDataFinished := TRUE;
               Error := ADSWrite.ErrId;
           ELSE
               WriteState := 1;
           END_IF
        ELSE
           ADSWrite(
               NETID:= '',
               PORT:= stCANopenDevice.PortNr,
               IDXGRP:= CO_Index,
               IDXOFFS:= CO_SubIndex,
               LEN:= DataLength,
               SRCADDR:= ADR(WriteData),
               WRITE:= FALSE,
               TMOUT := T#1s
               );
        END_IF
    1:
        ADSWrite(WRITE:= FALSE);
        IF ADSWrite.err THEN
           WriteState := 2;
           WriteDataFinished := TRUE;
           Error := ADSWrite.ErrId;
        ELSE
           IF NOT ADSWrite.busy THEN
               WriteState := 2;
               WriteDataFinished := TRUE;
           END_IF
        END_IF
    2:
        ADSWrite(WRITE:= FALSE);
		bStartWriting := FALSE;
        WriteState := 0;
END_CASE

METHOD PUBLIC GetReadDataAsUDINT : UDINT
VAR
	temp : UDINT;
END_VAR
MEMCPY(destAddr:=ADR(temp), srcAddr:=ADR(ReadData), n:=SIZEOF(UDINT));
GetReadDataAsUDINT := temp;
END_METHOD

METHOD PUBLIC GetReadDataAsUSINT : USINT
VAR
	temp : USINT;
END_VAR
MEMCPY(destAddr:=ADR(temp), srcAddr:=ADR(ReadData), n:=SIZEOF(USINT));
GetReadDataAsUSINT := temp;
END_METHOD

METHOD PUBLIC SetWriteDataFromUDINT
VAR_INPUT
	data : UDINT;
END_VAR
MEMCPY(destAddr:=ADR(WriteData), srcAddr:=ADR(data), n:=SIZEOF(UDINT));
END_METHOD

METHOD PUBLIC SetWriteDataFromUSINT
VAR_INPUT
	data : USINT;
END_VAR
MEMCPY(destAddr:=ADR(WriteData), srcAddr:=ADR(data), n:=SIZEOF(USINT));
END_METHOD

END_FUNCTION_BLOCK

// ---- POUs/FB_PDxxSimulation.TcPOU

FUNCTION_BLOCK FB_PDxxSimulation
VAR_INPUT
	Parameters								: ST_PDxx_SimulationParameters;
	RxPDO_1_6040h_ControlWord  				: UINT;
	RxPDO_1_6060h_ModesOfOperation  		: SINT;
	RxPDO_1_3202h_MotorDriveSubmodeSelect  	: UDINT;
	RxPDO_2_607Ah_TargetPosition  			: DINT;
	RxPDO_2_6081h_ProfileVelocity			: UDINT;
	RxPDO_3_6042h_TargetVelocity			: INT;
	RxPDO_4_60FEh_DigitalOutputs			: UDINT;

END_VAR
VAR_OUTPUT
	TxPDO_1_6041h_StatusWord  				: UINT;
	TxPDO_1_6061h_ModesOfOperationDisplay  	: SINT;
	TxPDO_2_6064h_PositionActualValue  		: DINT;
	TxPDO_3_6044h_VelocityActualValue  		: INT;
	TxPDO_4_60FDh_DigitalInputs  			: UDINT;

END_VAR
VAR
	stControlWord		: ST_PDxx_ControlWord;
	stStatusWord		: ST_PDxx_StatusWord;
	eTransition			: E_PDxx_TransitionCommand;
	trExecuteMove		: R_TRIG;
	bPositionMoveActive	: BOOL;
	nPosition			: LREAL;
	eState				: E_PDxx_State				:= E_PDxx_State.SWITCH_ON_DISABLED;
	eModesOfOperation	: E_PDxx_ModesOfOperation	:= E_PDxx_ModesOfOperation.NO_MODE_CHANGE_OR_NO_MODE_ASSIGNED;
END_VAR


A_ParseControlWord();
A_ParseTransition();
A_Motor();
A_SetStatusWord();

ACTION A_Motor:

IF eState = E_PDxx_State.OPERATION_ENABLED THEN
	CASE eModesOfOperation OF
		E_PDxx_ModesOfOperation.VELOCITY_MODE:
			VelocityMode();
		E_PDxx_ModesOfOperation.PROFILE_POSITION_MODE:
			ProfilePositionMode();
	END_CASE
ELSE
	TxPDO_3_6044h_VelocityActualValue := 0;
END_IF

TxPDO_2_6064h_PositionActualValue := LREAL_TO_DINT(nPosition);
END_ACTION

ACTION A_ParseControlWord:
 stControlWord.SwitchedOn_bit_0				:= RxPDO_1_6040h_ControlWord.0;
 stControlWord.EnableVoltage_bit_1			:= RxPDO_1_6040h_ControlWord.1;
 stControlWord.QuickStop_bit_2				:= RxPDO_1_6040h_ControlWord.2;
 stControlWord.EnableOperation_bit_3		:= RxPDO_1_6040h_ControlWord.3;
 stControlWord.OperationModeSpecific_bit_4	:= RxPDO_1_6040h_ControlWord.4;
 stControlWord.OperationModeSpecific_bit_5	:= RxPDO_1_6040h_ControlWord.5;
 stControlWord.OperationModeSpecific_bit_6	:= RxPDO_1_6040h_ControlWord.6;
 stControlWord.FaultReset_bit_7				:= RxPDO_1_6040h_ControlWord.7;
 stControlWord.Halt_bit_8					:= RxPDO_1_6040h_ControlWord.8;
 stControlWord.OperationModeSpecific_bit_9	:= RxPDO_1_6040h_ControlWord.9;
END_ACTION

ACTION A_ParseTransition:
IF
	stControlWord.FaultReset_bit_7 = TRUE AND
   	eTransition <> E_PDxx_TransitionCommand.FAULT_RESET THEN
		eTransition := E_PDxx_TransitionCommand.FAULT_RESET;
ELSIF
	stControlWord.SwitchedOn_bit_0 = FALSE AND
	stControlWord.EnableVoltage_bit_1 = TRUE AND
	stControlWord.QuickStop_bit_2 = TRUE AND
	stControlWord.FaultReset_bit_7 = FALSE THEN
		eTransition := E_PDxx_TransitionCommand.SHUTDOWN;
ELSIF
	stControlWord.SwitchedOn_bit_0 = TRUE AND
	stControlWord.EnableVoltage_bit_1 = TRUE AND
	stControlWord.QuickStop_bit_2 = TRUE AND
	stControlWord.EnableOperation_bit_3 = FALSE AND
	stControlWord.FaultReset_bit_7 = FALSE THEN
		eTransition := E_PDxx_TransitionCommand.SWITCH_ON;
ELSIF
	stControlWord.EnableVoltage_bit_1 = FALSE AND
	stControlWord.FaultReset_bit_7 = FALSE THEN
		eTransition := E_PDxx_TransitionCommand.DISABLE_VOLTAGE;
ELSIF
	stControlWord.EnableVoltage_bit_1 = TRUE AND
	stControlWord.QuickStop_bit_2 = FALSE AND
	stControlWord.FaultReset_bit_7 = FALSE THEN
		eTransition := E_PDxx_TransitionCommand.QUICK_STOP;
ELSIF
	stControlWord.SwitchedOn_bit_0 = TRUE AND
	stControlWord.EnableVoltage_bit_1 = TRUE AND
	stControlWord.QuickStop_bit_2 = TRUE AND
	stControlWord.EnableOperation_bit_3 = TRUE AND
	stControlWord.FaultReset_bit_7 = FALSE THEN
		eTransition := E_PDxx_TransitionCommand.ENABLE_OPERATION;
END_IF

CASE eTransition OF
	E_PDxx_TransitionCommand.FAULT_RESET:
		IF eState = E_PDxx_State.FAULT THEN
			eState := E_PDxx_State.SWITCH_ON_DISABLED;
		END_IF
	E_PDxx_TransitionCommand.SHUTDOWN:
		IF eState = E_PDxx_State.SWITCH_ON_DISABLED OR
		   eState = E_PDxx_State.SWITCHED_ON OR
		   eState = E_PDxx_State.OPERATION_ENABLED THEN
			eState := E_PDxx_State.READY_TO_SWITCH_ON;
		END_IF
	E_PDxx_TransitionCommand.SWITCH_ON:
		IF eState = E_PDxx_State.READY_TO_SWITCH_ON OR
		   eState = E_PDxx_State.OPERATION_ENABLED THEN
			eState := E_PDxx_State.SWITCHED_ON;
		END_IF
	E_PDxx_TransitionCommand.DISABLE_VOLTAGE:
		IF eState = E_PDxx_State.READY_TO_SWITCH_ON OR
		   eState = E_PDxx_State.SWITCHED_ON OR
		   eState = E_PDxx_State.OPERATION_ENABLED OR
		   eState = E_PDxx_State.QUICK_STOP_ACTIVE THEN
			eState := E_PDxx_State.SWITCH_ON_DISABLED;
		END_IF
	E_PDxx_TransitionCommand.QUICK_STOP:
		IF eState = E_PDxx_State.OPERATION_ENABLED THEN
			eState := E_PDxx_State.QUICK_STOP_ACTIVE;
		END_IF
	E_PDxx_TransitionCommand.ENABLE_OPERATION:
		IF eState = E_PDxx_State.SWITCHED_ON THEN
			eState := E_PDxx_State.OPERATION_ENABLED;
		END_IF
END_CASE

IF eState = E_PDxx_State.SWITCH_ON_DISABLED OR
   eState = E_PDxx_State.READY_TO_SWITCH_ON OR
   eState = E_PDxx_State.SWITCHED_ON THEN
   	TxPDO_1_6061h_ModesOfOperationDisplay := RxPDO_1_6060h_ModesOfOperation;
END_IF

CASE TxPDO_1_6061h_ModesOfOperationDisplay OF
	-2: eModesOfOperation := E_PDxx_ModesOfOperation.AUTO_SETUP;
	-1: eModesOfOperation := E_PDxx_ModesOfOperation.CLOCK_DIRECTION_MODE;
	0: eModesOfOperation := E_PDxx_ModesOfOperation.NO_MODE_CHANGE_OR_NO_MODE_ASSIGNED;
	1: eModesOfOperation := E_PDxx_ModesOfOperation.PROFILE_POSITION_MODE;
	2: eModesOfOperation := E_PDxx_ModesOfOperation.VELOCITY_MODE;
	3: eModesOfOperation := E_PDxx_ModesOfOperation.PROFILE_VELOCITY_MODE;
	4: eModesOfOperation := E_PDxx_ModesOfOperation.PROFILE_TORQUE_MODE;
	5: eModesOfOperation := E_PDxx_ModesOfOperation.RESERVED;
	6: eModesOfOperation := E_PDxx_ModesOfOperation.HOMING_MODE;
	7: eModesOfOperation := E_PDxx_ModesOfOperation.INTERPOLATED_POSITION_MODE;
	8: eModesOfOperation := E_PDxx_ModesOfOperation.CYCLIC_SYNCHRONOUS_POSITION_MODE;
	9: eModesOfOperation := E_PDxx_ModesOfOperation.CYCLIC_SYNCHRONOUS_VELOCITY_MODE;
	10: eModesOfOperation := E_PDxx_ModesOfOperation.CYCLIC_SYNCHRONOUS_TORQUE_MODE;	
END_CASE
END_ACTION

ACTION A_SetStatusWord:
CASE eState OF
	E_PDxx_State.NOT_READY_TO_SWITCH_ON:
		stStatusWord.ReadyToSwitchOn	:= FALSE;
		stStatusWord.SwitchedOn			:= FALSE;
		stStatusWord.OperationEnabled	:= FALSE;
		stStatusWord.Fault				:= FALSE;
//		stStatusWord.VoltageEnabled		:= FALSE;
//		stStatusWord.QuickStop			:= FALSE;
		stStatusWord.SwitchOnDisabled	:= FALSE;
	E_PDxx_State.SWITCH_ON_DISABLED:
		stStatusWord.ReadyToSwitchOn	:= FALSE;
		stStatusWord.SwitchedOn			:= FALSE;
		stStatusWord.OperationEnabled	:= FALSE;
		stStatusWord.Fault				:= FALSE;
//		stStatusWord.VoltageEnabled		:= FALSE;
//		stStatusWord.QuickStop			:= FALSE;
		stStatusWord.SwitchOnDisabled	:= TRUE;
	E_PDxx_State.READY_TO_SWITCH_ON:
		stStatusWord.ReadyToSwitchOn	:= TRUE;
		stStatusWord.SwitchedOn			:= FALSE;
		stStatusWord.OperationEnabled	:= FALSE;
		stStatusWord.Fault				:= FALSE;
//		stStatusWord.VoltageEnabled		:= FALSE;
		stStatusWord.QuickStop			:= TRUE;
		stStatusWord.SwitchOnDisabled	:= FALSE;
	E_PDxx_State.SWITCHED_ON:
		stStatusWord.ReadyToSwitchOn	:= TRUE;
		stStatusWord.SwitchedOn			:= TRUE;
		stStatusWord.OperationEnabled	:= FALSE;
		stStatusWord.Fault				:= FALSE;
//		stStatusWord.VoltageEnabled		:= FALSE;
		stStatusWord.QuickStop			:= TRUE;
		stStatusWord.SwitchOnDisabled	:= FALSE;
	E_PDxx_State.OPERATION_ENABLED:
		stStatusWord.ReadyToSwitchOn	:= TRUE;
		stStatusWord.SwitchedOn			:= TRUE;
		stStatusWord.OperationEnabled	:= TRUE;
		stStatusWord.Fault				:= FALSE;
//		stStatusWord.VoltageEnabled		:= FALSE;
		stStatusWord.QuickStop			:= TRUE;
		stStatusWord.SwitchOnDisabled	:= FALSE;
	E_PDxx_State.QUICK_STOP_ACTIVE:
		stStatusWord.ReadyToSwitchOn	:= TRUE;
		stStatusWord.SwitchedOn			:= TRUE;
		stStatusWord.OperationEnabled	:= TRUE;
		stStatusWord.Fault				:= FALSE;
//		stStatusWord.VoltageEnabled		:= FALSE;
		stStatusWord.QuickStop			:= FALSE;
		stStatusWord.SwitchOnDisabled	:= FALSE;
	E_PDxx_State.FAULT_REACTION_ACTIVE:
		stStatusWord.ReadyToSwitchOn	:= TRUE;
		stStatusWord.SwitchedOn			:= TRUE;
		stStatusWord.OperationEnabled	:= TRUE;
		stStatusWord.Fault				:= TRUE;
//		stStatusWord.VoltageEnabled		:= FALSE;
//		stStatusWord.QuickStop			:= FALSE;
		stStatusWord.SwitchOnDisabled	:= FALSE;
	E_PDxx_State.FAULT:
		stStatusWord.ReadyToSwitchOn	:= FALSE;
		stStatusWord.SwitchedOn			:= FALSE;
		stStatusWord.OperationEnabled	:= FALSE;
		stStatusWord.Fault				:= TRUE;
//		stStatusWord.VoltageEnabled		:= FALSE;
//		stStatusWord.QuickStop			:= FALSE;
		stStatusWord.SwitchOnDisabled	:= FALSE;
END_CASE

// Set more statusword bits if necessary for simulation, for example target reached and closed loop???

TxPDO_1_6041h_StatusWord.0 := stStatusWord.ReadyToSwitchOn;
TxPDO_1_6041h_StatusWord.1 := stStatusWord.SwitchedOn;
TxPDO_1_6041h_StatusWord.2 := stStatusWord.OperationEnabled;
TxPDO_1_6041h_StatusWord.3 := stStatusWord.Fault;
TxPDO_1_6041h_StatusWord.4 := stStatusWord.VoltageEnabled;
TxPDO_1_6041h_StatusWord.5 := stStatusWord.QuickStop;
TxPDO_1_6041h_StatusWord.6 := stStatusWord.SwitchOnDisabled;
TxPDO_1_6041h_StatusWord.7 := stStatusWord.Warning;
TxPDO_1_6041h_StatusWord.8 := stStatusWord.Synchronization;
TxPDO_1_6041h_StatusWord.9 := stStatusWord.Remote;
TxPDO_1_6041h_StatusWord.10 := stStatusWord.TargetReached;
TxPDO_1_6041h_StatusWord.11 := stStatusWord.InternalLimitReached;
TxPDO_1_6041h_StatusWord.12 := stStatusWord.OperationModeSpecific_bit12;
TxPDO_1_6041h_StatusWord.13 := stStatusWord.OperationModeSpecific_bit13;
TxPDO_1_6041h_StatusWord.15 := stStatusWord.ClosedLoopAvailable;
END_ACTION

METHOD PRIVATE ProfilePositionMode
VAR
	nDeltaPosition : LREAL;
	nTargetPosition : LREAL;
END_VAR
trExecuteMove(CLK := stControlWord.OperationModeSpecific_bit_4);
IF trExecuteMove.Q = TRUE THEN
	bPositionMoveActive := TRUE;
	stStatusWord.OperationModeSpecific_bit12 := TRUE;
END_IF

IF bPositionMoveActive = TRUE THEN
	nTargetPosition := DINT_TO_LREAL(RxPDO_2_607Ah_TargetPosition);
	stStatusWord.TargetReached := FALSE;

	IF nTargetPosition < nPosition THEN
		TxPDO_3_6044h_VelocityActualValue  := -UDINT_TO_INT(RxPDO_2_6081h_ProfileVelocity);
	ELSE
		TxPDO_3_6044h_VelocityActualValue  :=  UDINT_TO_INT(RxPDO_2_6081h_ProfileVelocity);
	END_IF
	
	nDeltaPosition := INT_TO_LREAL(TxPDO_3_6044h_VelocityActualValue) * Parameters.nMMPerSecondPerVelUnit * Parameters.nSecondsPerSimStep;

	IF nPosition < nTargetPosition AND
	   nPosition + nDeltaPosition >=  nTargetPosition THEN
		nPosition := nTargetPosition;
		TxPDO_3_6044h_VelocityActualValue := 0;
		stStatusWord.TargetReached := TRUE;
		bPositionMoveActive := FALSE;
		RETURN;
	END_IF
	
	IF nPosition > nTargetPosition AND
	   nPosition + nDeltaPosition <=  nTargetPosition THEN
		nPosition := nTargetPosition;
		TxPDO_3_6044h_VelocityActualValue := 0;
		stStatusWord.TargetReached := TRUE;
		bPositionMoveActive := FALSE;
		RETURN;
	END_IF
	
	nPosition := nPosition + nDeltaPosition; 
	
	IF nPosition < Parameters.nPositionMin THEN
		nPosition := Parameters.nPositionMin;
		TxPDO_3_6044h_VelocityActualValue := 0;
	END_IF
	
	IF nPosition > Parameters.nPositionMax THEN
		nPosition := Parameters.nPositionMax;
		TxPDO_3_6044h_VelocityActualValue := 0;
	END_IF

END_IF

IF stControlWord.OperationModeSpecific_bit_4 = FALSE THEN
	stStatusWord.OperationModeSpecific_bit12 := FALSE;
END_IF
END_METHOD


METHOD PRIVATE VelocityMode
VAR
	nInsertedObjectThickness : LREAL;
END_VAR

TxPDO_3_6044h_VelocityActualValue  :=  RxPDO_3_6042h_TargetVelocity;

nPosition := nPosition + DINT_TO_LREAL(TxPDO_3_6044h_VelocityActualValue) * Parameters.nMMPerSecondPerVelUnit * Parameters.nSecondsPerSimStep; 

IF Parameters.bObjectInserted = TRUE THEN
	nInsertedObjectThickness := Parameters.nObjectThickness;
END_IF

IF nPosition < Parameters.nPositionMin + nInsertedObjectThickness THEN
	nPosition := Parameters.nPositionMin + nInsertedObjectThickness;
	TxPDO_3_6044h_VelocityActualValue := 0;
END_IF

IF nPosition > Parameters.nPositionMax THEN
	nPosition := Parameters.nPositionMax;
	TxPDO_3_6044h_VelocityActualValue := 0;
END_IF
END_METHOD

END_FUNCTION_BLOCK
